# B&R Automation Studio project 8238 (part 2)

### IoMap.iom - APC2200/IoMap.iom
```iecst
(********************************************************************
 * COPYRIGHT --
 ********************************************************************
 * File: IoMap.iom
 * Author: Dave
 * Created: November 19, 2010
 ********************************************************************
 * IO mapping file
 ********************************************************************)
VAR_CONFIG
	Safety.ModuleOk AT %IX."X20SL8100".ModuleOk;
	Safety.ModuleID AT %ID."X20SL8100".ModuleID;
	Safety.FW_Version AT %ID."X20SL8100".FirmwareVersion;
	Safety.SFW_Version AT %IW."X20SL8100".SafeFirmwareVersion;
	Safety.UDID_low AT %ID."X20SL8100".UDID_low;
	Safety.UDID_high AT %IW."X20SL8100".UDID_high;
	Safety.EDM_Comm AT %QD."X20SL8100".DINT101;
	Safety.Reset_Comm AT %QD."X20SL8100".DINT102;
	Safety.MasterReset_Comm AT %QW."X20SL8100".INT1001;
	Safety.ModuleFault AT %IX."X20SL8100".BOOL00001;
	SafetyZone[1].DataFromSafePLC AT %IW."X20SL8100".INT0001;
	SafetyZone[2].DataFromSafePLC AT %IW."X20SL8100".INT0002;
	SafetyZone[3].DataFromSafePLC AT %IW."X20SL8100".INT0003;
	SafetyZone[4].DataFromSafePLC AT %IW."X20SL8100".INT0004;
	SafetyZone[5].DataFromSafePLC AT %IW."X20SL8100".INT0005;
	SafetyZone[6].DataFromSafePLC AT %IW."X20SL8100".INT0006;
	SafetyZone[7].DataFromSafePLC AT %IW."X20SL8100".INT0007;
	SafetyZone[8].DataFromSafePLC AT %IW."X20SL8100".INT0008;
	SafetyZone[9].DataFromSafePLC AT %IW."X20SL8100".INT0009;
	SafetyZone[10].DataFromSafePLC AT %IW."X20SL8100".INT0010;
	SafetyZone[11].DataFromSafePLC AT %IW."X20SL8100".INT0011;
	SafetyZone[12].DataFromSafePLC AT %IW."X20SL8100".INT0012;
	SafetyZone[13].DataFromSafePLC AT %IW."X20SL8100".INT0013;
	SafetyZone[14].DataFromSafePLC AT %IW."X20SL8100".INT0014;
	SafetyZone[15].DataFromSafePLC AT %IW."X20SL8100".INT0015;
	SafetyZone[16].DataFromSafePLC AT %IW."X20SL8100".INT0016;
	SafetyZone[17].DataFromSafePLC AT %IW."X20SL8100".INT0017;
	SafetyZone[18].DataFromSafePLC AT %IW."X20SL8100".INT0018;
	SafetyZone[19].DataFromSafePLC AT %IW."X20SL8100".INT0019;
	SafetyZone[20].DataFromSafePLC AT %IW."X20SL8100".INT0020;
	SafetyZone[21].DataFromSafePLC AT %IW."X20SL8100".INT0021;
	SafetyZone[22].DataFromSafePLC AT %IW."X20SL8100".INT0022;
	SafetyZone[23].DataFromSafePLC AT %IW."X20SL8100".INT0023;
	SafetyZone[24].DataFromSafePLC AT %IW."X20SL8100".INT0024;
	SafetyZone[25].DataFromSafePLC AT %IW."X20SL8100".INT0025;
	SafetyZone[26].DataFromSafePLC AT %IW."X20SL8100".INT0026;
	SafetyZone[27].DataFromSafePLC AT %IW."X20SL8100".INT0027;
	SafetyZone[28].DataFromSafePLC AT %IW."X20SL8100".INT0028;
	SafetyZone[29].DataFromSafePLC AT %IW."X20SL8100".INT0029;
	SafetyZone[30].DataFromSafePLC AT %IW."X20SL8100".INT0030;
	Safety.EDM_Comm AT %QD."X20SL8100".DINT1001;
	Safety.Reset_Comm AT %QD."X20SL8100".DINT1002;
	Cyclic#2.OK[1001] AT %IX."X20DM9324_1001".ModuleOk;
	Cyclic#2.OK[1002] AT %IX."X20DM9324_1002".ModuleOk;
	BusCouplerDiag[21].ModuleLostWhilstOperational AT %ID."X20BB80_400_MC01".IF1.ModuleLostWhileOperational;
	BusCouplerDiag[21].StationAtBusEnd AT %IB."X20BB80_400_MC01".IF1.StationAtBusEnd;
	BusCouplerDiag[21].StationPastOutFrameError AT %IB."X20BB80_400_MC01".IF1.StationPastOutFrameError;
	BusCouplerDiag[21].StationPastInFrameError AT %IB."X20BB80_400_MC01".IF1.StationPastInFrameError;
	BusCouplerDiag[31].ModuleLostWhilstOperational AT %ID."X67BC8321_PL31".IF1.ModuleLostWhileOperational;
	BusCouplerDiag[31].StationAtBusEnd AT %IB."X67BC8321_PL31".IF1.StationAtBusEnd;
	BusCouplerDiag[31].StationPastOutFrameError AT %IB."X67BC8321_PL31".IF1.StationPastOutFrameError;
	BusCouplerDiag[31].StationPastInFrameError AT %IB."X67BC8321_PL31".IF1.StationPastInFrameError;
	BusCouplerDiag[32].ModuleLostWhilstOperational AT %ID."X67BC8321_PL32".IF1.ModuleLostWhileOperational;
	BusCouplerDiag[32].StationAtBusEnd AT %IB."X67BC8321_PL32".IF1.StationAtBusEnd;
	BusCouplerDiag[32].StationPastOutFrameError AT %IB."X67BC8321_PL32".IF1.StationPastOutFrameError;
	BusCouplerDiag[32].StationPastInFrameError AT %IB."X67BC8321_PL32".IF1.StationPastInFrameError;
	BusCouplerDiag[33].ModuleLostWhilstOperational AT %ID."X67BC8321_PL33".IF1.ModuleLostWhileOperational;
	BusCouplerDiag[33].StationAtBusEnd AT %IB."X67BC8321_PL33".IF1.StationAtBusEnd;
	BusCouplerDiag[33].StationPastOutFrameError AT %IB."X67BC8321_PL33".IF1.StationPastOutFrameError;
	BusCouplerDiag[33].StationPastInFrameError AT %IB."X67BC8321_PL33".IF1.StationPastInFrameError;
	BusCouplerDiag[110].ModuleLostWhilstOperational AT %ID."X20BB80_400_SC01".IF1.ModuleLostWhileOperational;
	BusCouplerDiag[110].StationAtBusEnd AT %IB."X20BB80_400_SC01".IF1.StationAtBusEnd;
	BusCouplerDiag[110].StationPastOutFrameError AT %IB."X20BB80_400_SC01".IF1.StationPastOutFrameError;
	BusCouplerDiag[110].StationPastInFrameError AT %IB."X20BB80_400_SC01".IF1.StationPastInFrameError;
	Cyclic#2.ABB_EPL.Drives[11].Comm.ModuleOk AT %IX."FEPL-02_and_ACS380_SB1".ModuleOk;
	Cyclic#2.ABB_EPL.Drives[11].Comm.ErrorCode AT %IW."FEPL-02_and_ACS380_SB1".VendorSpecificAlarmCodes_I2203;
	Cyclic#2.ABB_EPL.Drives[11].Comm.ControlWord AT %QW."FEPL-02_and_ACS380_SB1".ControlWord_I6040Out;
	Cyclic#2.ABB_EPL.Drives[11].Comm.StatusWord AT %IW."FEPL-02_and_ACS380_SB1".StatusWord_I6041;
	Cyclic#2.ABB_EPL.Drives[11].Comm.TargetVelocity AT %QW."FEPL-02_and_ACS380_SB1".VlTargetVelocity_I6042Out;
	Cyclic#2.ABB_EPL.Drives[11].Comm.ActVelocity AT %IW."FEPL-02_and_ACS380_SB1".VlVelocityActualValue_I6044;
	Cyclic#2.ABB_EPL.Drives[11].Comm.ActCurrent AT %ID."FEPL-02_and_ACS380_SB1"._0107_Motor_current_I4001_S07;
	Cyclic#2.ABB_EPL.Drives[11].Comm.ActTorque AT %ID."FEPL-02_and_ACS380_SB1"._0110_Motor_torque_I4001_S0A;
	Cyclic#2.ABB_EPL.Drives[1].Comm.ModuleOk AT %IX."FEPL-02_and_ACS380_STB1".ModuleOk;
	Cyclic#2.ABB_EPL.Drives[1].Comm.ErrorCode AT %IW."FEPL-02_and_ACS380_STB1".VendorSpecificAlarmCodes_I2203;
	Cyclic#2.ABB_EPL.Drives[1].Comm.ControlWord AT %QW."FEPL-02_and_ACS380_STB1".ControlWord_I6040Out;
	Cyclic#2.ABB_EPL.Drives[1].Comm.StatusWord AT %IW."FEPL-02_and_ACS380_STB1".StatusWord_I6041;
	Cyclic#2.ABB_EPL.Drives[1].Comm.TargetVelocity AT %QW."FEPL-02_and_ACS380_STB1".VlTargetVelocity_I6042Out;
	Cyclic#2.ABB_EPL.Drives[1].Comm.ActVelocity AT %IW."FEPL-02_and_ACS380_STB1".VlVelocityActualValue_I6044;
	Cyclic#2.ABB_EPL.Drives[1].Comm.ActCurrent AT %ID."FEPL-02_and_ACS380_STB1"._0107_Motor_current_I4001_S07;
	Cyclic#2.ABB_EPL.Drives[1].Comm.ActTorque AT %ID."FEPL-02_and_ACS380_STB1"._0110_Motor_torque_I4001_S0A;
	Cyclic#2.ABB_EPL.Drives[12].Comm.ModuleOk AT %IX."FEPL-02_and_ACS380_SB2".ModuleOk;
	Cyclic#2.ABB_EPL.Drives[12].Comm.ErrorCode AT %IW."FEPL-02_and_ACS380_SB2".VendorSpecificAlarmCodes_I2203;
	Cyclic#2.ABB_EPL.Drives[12].Comm.ControlWord AT %QW."FEPL-02_and_ACS380_SB2".ControlWord_I6040Out;
	Cyclic#2.ABB_EPL.Drives[12].Comm.StatusWord AT %IW."FEPL-02_and_ACS380_SB2".StatusWord_I6041;
	Cyclic#2.ABB_EPL.Drives[12].Comm.TargetVelocity AT %QW."FEPL-02_and_ACS380_SB2".VlTargetVelocity_I6042Out;
	Cyclic#2.ABB_EPL.Drives[12].Comm.ActVelocity AT %IW."FEPL-02_and_ACS380_SB2".VlVelocityActualValue_I6044;
	Cyclic#2.ABB_EPL.Drives[12].Comm.ActCurrent AT %ID."FEPL-02_and_ACS380_SB2"._0107_Motor_current_I4001_S07;
	Cyclic#2.ABB_EPL.Drives[12].Comm.ActTorque AT %ID."FEPL-02_and_ACS380_SB2"._0110_Motor_torque_I4001_S0A;
	Cyclic#2.ABB_EPL.Drives[2].Comm.ModuleOk AT %IX."FEPL-02_and_ACS380_STB2".ModuleOk;
	Cyclic#2.ABB_EPL.Drives[2].Comm.ErrorCode AT %IW."FEPL-02_and_ACS380_STB2".VendorSpecificAlarmCodes_I2203;
	Cyclic#2.ABB_EPL.Drives[2].Comm.ControlWord AT %QW."FEPL-02_and_ACS380_STB2".ControlWord_I6040Out;
	Cyclic#2.ABB_EPL.Drives[2].Comm.StatusWord AT %IW."FEPL-02_and_ACS380_STB2".StatusWord_I6041;
	Cyclic#2.ABB_EPL.Drives[2].Comm.TargetVelocity AT %QW."FEPL-02_and_ACS380_STB2".VlTargetVelocity_I6042Out;
	Cyclic#2.ABB_EPL.Drives[2].Comm.ActVelocity AT %IW."FEPL-02_and_ACS380_STB2".VlVelocityActualValue_I6044;
	Cyclic#2.ABB_EPL.Drives[2].Comm.ActCurrent AT %ID."FEPL-02_and_ACS380_STB2"._0107_Motor_current_I4001_S07;
	Cyclic#2.ABB_EPL.Drives[2].Comm.ActTorque AT %ID."FEPL-02_and_ACS380_STB2"._0110_Motor_torque_I4001_S0A;
	SM[1401].ModuleOk AT %IX."X67SI8103_1401".ModuleOk;
	SM[1401].ModuleID AT %IW."X67SI8103_1401".ModuleID;
	SM[1401].HardwareVariant AT %IW."X67SI8103_1401".HardwareVariant;
	SM[1401].FirmwareVersion AT %IW."X67SI8103_1401".FirmwareVersion;
	SM[1401].SafeModuleOK AT %IX."X67SI8103_1401".SafeModuleOK;
	SM[1401].SafeDigitialInput01 AT %IX."X67SI8103_1401".SafeDigitalInput01;
	SM[1401].SafeDigitialInput02 AT %IX."X67SI8103_1401".SafeDigitalInput02;
	SM[1401].SafeDigitialInput03 AT %IX."X67SI8103_1401".SafeDigitalInput03;
	SM[1401].SafeDigitialInput04 AT %IX."X67SI8103_1401".SafeDigitalInput04;
	SM[1401].SafeDigitialInput05 AT %IX."X67SI8103_1401".SafeDigitalInput05;
	SM[1401].SafeDigitialInput06 AT %IX."X67SI8103_1401".SafeDigitalInput06;
	SM[1401].SafeDigitialInput07 AT %IX."X67SI8103_1401".SafeDigitalInput07;
	SM[1401].SafeDigitialInput08 AT %IX."X67SI8103_1401".SafeDigitalInput08;
	SM[1401].SafeTwoChannelInput0102 AT %IX."X67SI8103_1401".SafeTwoChannelInput0102;
	SM[1401].SafeTwoChannelInput0304 AT %IX."X67SI8103_1401".SafeTwoChannelInput0304;
	SM[1401].SafeTwoChannelInput0506 AT %IX."X67SI8103_1401".SafeTwoChannelInput0506;
	SM[1401].SafeTwoChannelInput0708 AT %IX."X67SI8103_1401".SafeTwoChannelInput0708;
	SM[1401].SafeTwoChannelOk0102 AT %IX."X67SI8103_1401".SafeTwoChannelOK0102;
	SM[1401].SafeTwoChannelOk0304 AT %IX."X67SI8103_1401".SafeTwoChannelOK0304;
	SM[1401].SafeTwoChannelOk0506 AT %IX."X67SI8103_1401".SafeTwoChannelOK0506;
	SM[1401].SafeTwoChannelOk0708 AT %IX."X67SI8103_1401".SafeTwoChannelOK0708;
	SM[1401].DigitalInput01 AT %IX."X67SI8103_1401".DigitalInput01;
	SM[1401].DigitalInput02 AT %IX."X67SI8103_1401".DigitalInput02;
	SM[1401].DigitalOutput01 AT %QX."X67SI8103_1401".DigitalOutput01;
	SM[1401].DigitalOutput02 AT %QX."X67SI8103_1401".DigitalOutput02;
	SM[1402].ModuleOk AT %IX."X67SI8103_1402".ModuleOk;
	SM[1402].ModuleID AT %IW."X67SI8103_1402".ModuleID;
	SM[1402].HardwareVariant AT %IW."X67SI8103_1402".HardwareVariant;
	SM[1402].FirmwareVersion AT %IW."X67SI8103_1402".FirmwareVersion;
	SM[1402].SafeModuleOK AT %IX."X67SI8103_1402".SafeModuleOK;
	SM[1402].SafeDigitialInput01 AT %IX."X67SI8103_1402".SafeDigitalInput01;
	SM[1402].SafeDigitialInput02 AT %IX."X67SI8103_1402".SafeDigitalInput02;
	SM[1402].SafeDigitialInput03 AT %IX."X67SI8103_1402".SafeDigitalInput03;
	SM[1402].SafeDigitialInput04 AT %IX."X67SI8103_1402".SafeDigitalInput04;
	SM[1402].SafeDigitialInput05 AT %IX."X67SI8103_1402".SafeDigitalInput05;
	SM[1402].SafeDigitialInput06 AT %IX."X67SI8103_1402".SafeDigitalInput06;
	SM[1402].SafeDigitialInput07 AT %IX."X67SI8103_1402".SafeDigitalInput07;
	SM[1402].SafeDigitialInput08 AT %IX."X67SI8103_1402".SafeDigitalInput08;
	SM[1402].SafeTwoChannelInput0102 AT %IX."X67SI8103_1402".SafeTwoChannelInput0102;
	SM[1402].SafeTwoChannelInput0304 AT %IX."X67SI8103_1402".SafeTwoChannelInput0304;
	SM[1402].SafeTwoChannelInput0506 AT %IX."X67SI8103_1402".SafeTwoChannelInput0506;
	SM[1402].SafeTwoChannelInput0708 AT %IX."X67SI8103_1402".SafeTwoChannelInput0708;
	SM[1402].SafeTwoChannelOk0102 AT %IX."X67SI8103_1402".SafeTwoChannelOK0102;
	SM[1402].SafeTwoChannelOk0304 AT %IX."X67SI8103_1402".SafeTwoChannelOK0304;
	SM[1402].SafeTwoChannelOk0506 AT %IX."X67SI8103_1402".SafeTwoChannelOK0506;
	SM[1402].SafeTwoChannelOk0708 AT %IX."X67SI8103_1402".SafeTwoChannelOK0708;
	SM[1402].DigitalInput01 AT %IX."X67SI8103_1402".DigitalInput01;
	SM[1402].DigitalInput02 AT %IX."X67SI8103_1402".DigitalInput02;
	SM[1402].DigitalOutput01 AT %QX."X67SI8103_1402".DigitalOutput01;
	SM[1402].DigitalOutput02 AT %QX."X67SI8103_1402".DigitalOutput02;
	SM[1403].ModuleOk AT %IX."X67SI8103_1403".ModuleOk;
	SM[1403].ModuleID AT %IW."X67SI8103_1403".ModuleID;
	SM[1403].HardwareVariant AT %IW."X67SI8103_1403".HardwareVariant;
	SM[1403].FirmwareVersion AT %IW."X67SI8103_1403".FirmwareVersion;
	SM[1403].SafeModuleOK AT %IX."X67SI8103_1403".SafeModuleOK;
	SM[1403].SafeDigitialInput01 AT %IX."X67SI8103_1403".SafeDigitalInput01;
	SM[1403].SafeDigitialInput02 AT %IX."X67SI8103_1403".SafeDigitalInput02;
	SM[1403].SafeDigitialInput03 AT %IX."X67SI8103_1403".SafeDigitalInput03;
	SM[1403].SafeDigitialInput04 AT %IX."X67SI8103_1403".SafeDigitalInput04;
	SM[1403].SafeDigitialInput05 AT %IX."X67SI8103_1403".SafeDigitalInput05;
	SM[1403].SafeDigitialInput06 AT %IX."X67SI8103_1403".SafeDigitalInput06;
	SM[1403].SafeDigitialInput07 AT %IX."X67SI8103_1403".SafeDigitalInput07;
	SM[1403].SafeDigitialInput08 AT %IX."X67SI8103_1403".SafeDigitalInput08;
	SM[1403].SafeTwoChannelInput0102 AT %IX."X67SI8103_1403".SafeTwoChannelInput0102;
	SM[1403].SafeTwoChannelInput0304 AT %IX."X67SI8103_1403".SafeTwoChannelInput0304;
	SM[1403].SafeTwoChannelInput0506 AT %IX."X67SI8103_1403".SafeTwoChannelInput0506;
	SM[1403].SafeTwoChannelInput0708 AT %IX."X67SI8103_1403".SafeTwoChannelInput0708;
	SM[1403].SafeTwoChannelOk0102 AT %IX."X67SI8103_1403".SafeTwoChannelOK0102;
	SM[1403].SafeTwoChannelOk0304 AT %IX."X67SI8103_1403".SafeTwoChannelOK0304;
	SM[1403].SafeTwoChannelOk0506 AT %IX."X67SI8103_1403".SafeTwoChannelOK0506;
	SM[1403].SafeTwoChannelOk0708 AT %IX."X67SI8103_1403".SafeTwoChannelOK0708;
	SM[1403].DigitalInput01 AT %IX."X67SI8103_1403".DigitalInput01;
	SM[1403].DigitalInput02 AT %IX."X67SI8103_1403".DigitalInput02;
	SM[1403].DigitalOutput01 AT %QX."X67SI8103_1403".DigitalOutput01;
	SM[1403].DigitalOutput02 AT %QX."X67SI8103_1403".DigitalOutput02;
	SM[1406].ModuleOk AT %IX."X67SI8103_1406".ModuleOk;
	SM[1406].ModuleID AT %IW."X67SI8103_1406".ModuleID;
	SM[1406].HardwareVariant AT %IW."X67SI8103_1406".HardwareVariant;
	SM[1406].FirmwareVersion AT %IW."X67SI8103_1406".FirmwareVersion;
	SM[1406].SafeModuleOK AT %IX."X67SI8103_1406".SafeModuleOK;
	SM[1406].SafeDigitialInput01 AT %IX."X67SI8103_1406".SafeDigitalInput01;
	SM[1406].SafeDigitialInput02 AT %IX."X67SI8103_1406".SafeDigitalInput02;
	SM[1406].SafeDigitialInput03 AT %IX."X67SI8103_1406".SafeDigitalInput03;
	SM[1406].SafeDigitialInput04 AT %IX."X67SI8103_1406".SafeDigitalInput04;
	SM[1406].SafeDigitialInput05 AT %IX."X67SI8103_1406".SafeDigitalInput05;
	SM[1406].SafeDigitialInput06 AT %IX."X67SI8103_1406".SafeDigitalInput06;
	SM[1406].SafeDigitialInput07 AT %IX."X67SI8103_1406".SafeDigitalInput07;
	SM[1406].SafeDigitialInput08 AT %IX."X67SI8103_1406".SafeDigitalInput08;
	SM[1406].SafeTwoChannelInput0102 AT %IX."X67SI8103_1406".SafeTwoChannelInput0102;
	SM[1406].SafeTwoChannelInput0304 AT %IX."X67SI8103_1406".SafeTwoChannelInput0304;
	SM[1406].SafeTwoChannelInput0506 AT %IX."X67SI8103_1406".SafeTwoChannelInput0506;
	SM[1406].SafeTwoChannelInput0708 AT %IX."X67SI8103_1406".SafeTwoChannelInput0708;
	SM[1406].SafeTwoChannelOk0102 AT %IX."X67SI8103_1406".SafeTwoChannelOK0102;
	SM[1406].SafeTwoChannelOk0304 AT %IX."X67SI8103_1406".SafeTwoChannelOK0304;
	SM[1406].SafeTwoChannelOk0506 AT %IX."X67SI8103_1406".SafeTwoChannelOK0506;
	SM[1406].SafeTwoChannelOk0708 AT %IX."X67SI8103_1406".SafeTwoChannelOK0708;
	SM[1406].DigitalInput01 AT %IX."X67SI8103_1406".DigitalInput01;
	SM[1406].DigitalInput02 AT %IX."X67SI8103_1406".DigitalInput02;
	SM[1406].DigitalOutput01 AT %QX."X67SI8103_1406".DigitalOutput01;
	SM[1406].DigitalOutput02 AT %QX."X67SI8103_1406".DigitalOutput02;
	WeightRaw[1349].Wgt_Channel_1 AT %ID."X67AI2744_1801".AnalogInput01;
	WeightRaw[1352].Wgt_Channel_1 AT %ID."X67AI2744_1802".AnalogInput01;
	WeightRaw[1355].Wgt_Channel_1 AT %ID."X67AI2744_1803".AnalogInput01;
	SM[1410].ModuleOk AT %IX."X67SI8103_1410".ModuleOk;
	SM[1410].ModuleID AT %IW."X67SI8103_1410".ModuleID;
	SM[1410].HardwareVariant AT %IW."X67SI8103_1410".HardwareVariant;
	SM[1410].FirmwareVersion AT %IW."X67SI8103_1410".FirmwareVersion;
	SM[1410].SafeModuleOK AT %IX."X67SI8103_1410".SafeModuleOK;
	SM[1410].SafeDigitialInput01 AT %IX."X67SI8103_1410".SafeDigitalInput01;
	SM[1410].SafeDigitialInput02 AT %IX."X67SI8103_1410".SafeDigitalInput02;
	SM[1410].SafeDigitialInput03 AT %IX."X67SI8103_1410".SafeDigitalInput03;
	SM[1410].SafeDigitialInput04 AT %IX."X67SI8103_1410".SafeDigitalInput04;
	SM[1410].SafeDigitialInput05 AT %IX."X67SI8103_1410".SafeDigitalInput05;
	SM[1410].SafeDigitialInput06 AT %IX."X67SI8103_1410".SafeDigitalInput06;
	SM[1410].SafeDigitialInput07 AT %IX."X67SI8103_1410".SafeDigitalInput07;
	SM[1410].SafeDigitialInput08 AT %IX."X67SI8103_1410".SafeDigitalInput08;
	SM[1410].SafeTwoChannelInput0102 AT %IX."X67SI8103_1410".SafeTwoChannelInput0102;
	SM[1410].SafeTwoChannelInput0304 AT %IX."X67SI8103_1410".SafeTwoChannelInput0304;
	SM[1410].SafeTwoChannelInput0506 AT %IX."X67SI8103_1410".SafeTwoChannelInput0506;
	SM[1410].SafeTwoChannelInput0708 AT %IX."X67SI8103_1410".SafeTwoChannelInput0708;
	SM[1410].SafeTwoChannelOk0102 AT %IX."X67SI8103_1410".SafeTwoChannelOK0102;
	SM[1410].SafeTwoChannelOk0304 AT %IX."X67SI8103_1410".SafeTwoChannelOK0304;
	SM[1410].SafeTwoChannelOk0506 AT %IX."X67SI8103_1410".SafeTwoChannelOK0506;
	SM[1410].SafeTwoChannelOk0708 AT %IX."X67SI8103_1410".SafeTwoChannelOK0708;
	SM[1410].DigitalInput01 AT %IX."X67SI8103_1410".DigitalInput01;
	SM[1410].DigitalInput02 AT %IX."X67SI8103_1410".DigitalInput02;
	SM[1410].DigitalOutput01 AT %QX."X67SI8103_1410".DigitalOutput01;
	SM[1410].DigitalOutput02 AT %QX."X67SI8103_1410".DigitalOutput02;
	SM[1411].ModuleOk AT %IX."X67SI8103_1411".ModuleOk;
	SM[1411].ModuleID AT %IW."X67SI8103_1411".ModuleID;
	SM[1411].HardwareVariant AT %IW."X67SI8103_1411".HardwareVariant;
	SM[1411].FirmwareVersion AT %IW."X67SI8103_1411".FirmwareVersion;
	SM[1411].SafeModuleOK AT %IX."X67SI8103_1411".SafeModuleOK;
	SM[1411].SafeDigitialInput01 AT %IX."X67SI8103_1411".SafeDigitalInput01;
	SM[1411].SafeDigitialInput02 AT %IX."X67SI8103_1411".SafeDigitalInput02;
	SM[1411].SafeDigitialInput03 AT %IX."X67SI8103_1411".SafeDigitalInput03;
	SM[1411].SafeDigitialInput04 AT %IX."X67SI8103_1411".SafeDigitalInput04;
	SM[1411].SafeDigitialInput05 AT %IX."X67SI8103_1411".SafeDigitalInput05;
	SM[1411].SafeDigitialInput06 AT %IX."X67SI8103_1411".SafeDigitalInput06;
	SM[1411].SafeDigitialInput07 AT %IX."X67SI8103_1411".SafeDigitalInput07;
	SM[1411].SafeDigitialInput08 AT %IX."X67SI8103_1411".SafeDigitalInput08;
	SM[1411].SafeTwoChannelInput0102 AT %IX."X67SI8103_1411".SafeTwoChannelInput0102;
	SM[1411].SafeTwoChannelInput0304 AT %IX."X67SI8103_1411".SafeTwoChannelInput0304;
	SM[1411].SafeTwoChannelInput0506 AT %IX."X67SI8103_1411".SafeTwoChannelInput0506;
	SM[1411].SafeTwoChannelInput0708 AT %IX."X67SI8103_1411".SafeTwoChannelInput0708;
	SM[1411].SafeTwoChannelOk0102 AT %IX."X67SI8103_1411".SafeTwoChannelOK0102;
	SM[1411].SafeTwoChannelOk0304 AT %IX."X67SI8103_1411".SafeTwoChannelOK0304;
	SM[1411].SafeTwoChannelOk0506 AT %IX."X67SI8103_1411".SafeTwoChannelOK0506;
	SM[1411].SafeTwoChannelOk0708 AT %IX."X67SI8103_1411".SafeTwoChannelOK0708;
	SM[1411].DigitalInput01 AT %IX."X67SI8103_1411".DigitalInput01;
	SM[1411].DigitalInput02 AT %IX."X67SI8103_1411".DigitalInput02;
	SM[1411].DigitalOutput01 AT %QX."X67SI8103_1411".DigitalOutput01;
	SM[1411].DigitalOutput02 AT %QX."X67SI8103_1411".DigitalOutput02;
	SM[1416].ModuleOk AT %IX."X67SI8103_1416".ModuleOk;
	SM[1416].ModuleID AT %IW."X67SI8103_1416".ModuleID;
	SM[1416].HardwareVariant AT %IW."X67SI8103_1416".HardwareVariant;
	SM[1416].FirmwareVersion AT %IW."X67SI8103_1416".FirmwareVersion;
	SM[1416].SafeModuleOK AT %IX."X67SI8103_1416".SafeModuleOK;
	SM[1416].SafeDigitialInput01 AT %IX."X67SI8103_1416".SafeDigitalInput01;
	SM[1416].SafeDigitialInput02 AT %IX."X67SI8103_1416".SafeDigitalInput02;
	SM[1416].SafeDigitialInput03 AT %IX."X67SI8103_1416".SafeDigitalInput03;
	SM[1416].SafeDigitialInput04 AT %IX."X67SI8103_1416".SafeDigitalInput04;
	SM[1416].SafeDigitialInput05 AT %IX."X67SI8103_1416".SafeDigitalInput05;
	SM[1416].SafeDigitialInput06 AT %IX."X67SI8103_1416".SafeDigitalInput06;
	SM[1416].SafeDigitialInput07 AT %IX."X67SI8103_1416".SafeDigitalInput07;
	SM[1416].SafeDigitialInput08 AT %IX."X67SI8103_1416".SafeDigitalInput08;
	SM[1416].SafeTwoChannelInput0102 AT %IX."X67SI8103_1416".SafeTwoChannelInput0102;
	SM[1416].SafeTwoChannelInput0304 AT %IX."X67SI8103_1416".SafeTwoChannelInput0304;
	SM[1416].SafeTwoChannelInput0506 AT %IX."X67SI8103_1416".SafeTwoChannelInput0506;
	SM[1416].SafeTwoChannelInput0708 AT %IX."X67SI8103_1416".SafeTwoChannelInput0708;
	SM[1416].SafeTwoChannelOk0102 AT %IX."X67SI8103_1416".SafeTwoChannelOK0102;
	SM[1416].SafeTwoChannelOk0304 AT %IX."X67SI8103_1416".SafeTwoChannelOK0304;
	SM[1416].SafeTwoChannelOk0506 AT %IX."X67SI8103_1416".SafeTwoChannelOK0506;
	SM[1416].SafeTwoChannelOk0708 AT %IX."X67SI8103_1416".SafeTwoChannelOK0708;
	SM[1416].DigitalInput01 AT %IX."X67SI8103_1416".DigitalInput01;
	SM[1416].DigitalInput02 AT %IX."X67SI8103_1416".DigitalInput02;
	SM[1416].DigitalOutput01 AT %QX."X67SI8103_1416".DigitalOutput01;
	SM[1416].DigitalOutput02 AT %QX."X67SI8103_1416".DigitalOutput02;
	BusCouplerDiag[34].ModuleLostWhilstOperational AT %ID."X67BC8321_PL34".IF1.ModuleLostWhileOperational;
	BusCouplerDiag[34].StationAtBusEnd AT %IB."X67BC8321_PL34".IF1.StationAtBusEnd;
	BusCouplerDiag[34].StationPastOutFrameError AT %IB."X67BC8321_PL34".IF1.StationPastOutFrameError;
	BusCouplerDiag[34].StationPastInFrameError AT %IB."X67BC8321_PL34".IF1.StationPastInFrameError;
	BusCouplerDiag[35].ModuleLostWhilstOperational AT %ID."X67BC8321_PL35".IF1.ModuleLostWhileOperational;
	BusCouplerDiag[35].StationAtBusEnd AT %IB."X67BC8321_PL35".IF1.StationAtBusEnd;
	BusCouplerDiag[35].StationPastOutFrameError AT %IB."X67BC8321_PL35".IF1.StationPastOutFrameError;
	BusCouplerDiag[35].StationPastInFrameError AT %IB."X67BC8321_PL35".IF1.StationPastInFrameError;
	BusCouplerDiag[41].ModuleLostWhilstOperational AT %ID."X67BC8321_PL36".IF1.ModuleLostWhileOperational;
	BusCouplerDiag[42].ModuleLostWhilstOperational AT %ID."X67BC8321_PL37".IF1.ModuleLostWhileOperational;
	BusCouplerDiag[43].ModuleLostWhilstOperational AT %ID."X67BC8321_PL38".IF1.ModuleLostWhileOperational;
	BusCouplerDiag[44].ModuleLostWhilstOperational AT %ID."X67BC8321_PL39".IF1.ModuleLostWhileOperational;
	BusCouplerDiag[41].StationAtBusEnd AT %IB."X67BC8321_PL36".IF1.StationAtBusEnd;
	BusCouplerDiag[42].StationAtBusEnd AT %IB."X67BC8321_PL37".IF1.StationAtBusEnd;
	BusCouplerDiag[41].StationPastOutFrameError AT %IB."X67BC8321_PL36".IF1.StationPastOutFrameError;
	BusCouplerDiag[42].StationPastOutFrameError AT %IB."X67BC8321_PL37".IF1.StationPastOutFrameError;
	BusCouplerDiag[42].StationPastInFrameError AT %IB."X67BC8321_PL37".IF1.StationPastInFrameError;
	BusCouplerDiag[41].StationPastInFrameError AT %IB."X67BC8321_PL36".IF1.StationPastInFrameError;
	BusCouplerDiag[44].StationPastInFrameError AT %IB."X67BC8321_PL39".IF1.StationPastInFrameError;
	BusCouplerDiag[44].StationPastOutFrameError AT %IB."X67BC8321_PL39".IF1.StationPastOutFrameError;
	BusCouplerDiag[44].StationAtBusEnd AT %IB."X67BC8321_PL39".IF1.StationAtBusEnd;
	BusCouplerDiag[43].StationAtBusEnd AT %IB."X67BC8321_PL38".IF1.StationAtBusEnd;
	BusCouplerDiag[43].StationPastOutFrameError AT %IB."X67BC8321_PL38".IF1.StationPastOutFrameError;
	BusCouplerDiag[43].StationPastInFrameError AT %IB."X67BC8321_PL38".IF1.StationPastInFrameError;
	Cyclic#2.X[1001].X01 AT %IX."X20DM9324_1001".DigitalInput01; (*spare*) (*spare*)
	Cyclic#2.Y[1001].Y01 AT %QX."X20DM9324_1001".DigitalOutput01; (*Light Tower Green*) (*SafetyZone[1].TowerLight.TL_DO_Green*)
	Cyclic#2.X[1001].X02 AT %IX."X20DM9324_1001".DigitalInput02; (*Air pressure switch*) (*SafetyZone[1].PressureSwitch*)
	Cyclic#2.Y[1001].Y02 AT %QX."X20DM9324_1001".DigitalOutput02; (*Light Tower Yellow*) (*SafetyZone[1].TowerLight.TL_DO_Yellow*)
	Cyclic#2.X[1001].X03 AT %IX."X20DM9324_1001".DigitalInput03; (*Safety Reset button*) (*MasterReset_1*)
	Cyclic#2.Y[1001].Y03 AT %QX."X20DM9324_1001".DigitalOutput03; (*Light Tower Red*) (*SafetyZone[1].TowerLight.TL_DO_Red*)
	Cyclic#2.X[1001].X04 AT %IX."X20DM9324_1001".DigitalInput04; (*Fuse Reset*) (*Fuse_Reset_1*)
	Cyclic#2.Y[1001].Y04 AT %QX."X20DM9324_1001".DigitalOutput04; (*Light Tower Siren*) (*SafetyZone[1].TowerLight.TL_DO_Sounder*)
	Cyclic#2.X[1001].X05 AT %IX."X20DM9324_1001".DigitalInput05; (*spare*) (*spare*)
	Cyclic#2.X[1001].X06 AT %IX."X20DM9324_1001".DigitalInput06; (*spare*) (*spare*)
	Cyclic#2.X[1001].X07 AT %IX."X20DM9324_1001".DigitalInput07; (*spare*) (*spare*)
	Cyclic#2.X[1001].X08 AT %IX."X20DM9324_1001".DigitalInput08; (*spare*) (*spare*)
	Cyclic#2.X[1002].X01 AT %IX."X20DM9324_1002".DigitalInput01; (*Safety Relay D1.1 Monitor*) (*SafetyZone[2].EDM*)
	Cyclic#2.Y[1002].Y01 AT %QX."X20DM9324_1002".DigitalOutput01; (*Safety Reset Button Lamp*) (*SafetyZone[1].Main_Lamp*)
	Cyclic#2.X[1002].X02 AT %IX."X20DM9324_1002".DigitalInput02; (*Safety Relay D2.1 Monitor*) (*SafetyZone[3].EDM*)
	Cyclic#2.Y[1002].Y02 AT %QX."X20DM9324_1002".DigitalOutput02; (*Fuse Reset Button*) (*Fuse_Lamp_1*)
	Cyclic#2.X[1002].X03 AT %IX."X20DM9324_1002".DigitalInput03; (*Safety Relay D3.1 Monitor*) (*SafetyZone[4].EDM*)
	Cyclic#2.Y[1002].Y03 AT %QX."X20DM9324_1002".DigitalOutput03; (*spare*) (*spare*)
	Cyclic#2.X[1002].X04 AT %IX."X20DM9324_1002".DigitalInput04; (*Safety Relay D4.1 Monitor*) (*SafetyZone[5].EDM*)
	Cyclic#2.Y[1002].Y04 AT %QX."X20DM9324_1002".DigitalOutput04; (*spare*) (*spare*)
	Cyclic#2.X[1002].X05 AT %IX."X20DM9324_1002".DigitalInput05; (*spare*) (*spare*)
	Cyclic#2.X[1002].X06 AT %IX."X20DM9324_1002".DigitalInput06; (*spare*) (*spare*)
	Cyclic#2.X[1002].X07 AT %IX."X20DM9324_1002".DigitalInput07; (*spare*) (*spare*)
	Cyclic#2.X[1002].X08 AT %IX."X20DM9324_1002".DigitalInput08; (*spare*) (*spare*)
	Cyclic#2.OK[1302] AT %IX."X67DM1321_1302".ModuleOk;
	Cyclic#2.OK[1304] AT %IX."X67DM1321_1304".ModuleOk;
	Cyclic#2.OK[1306] AT %IX."X67DM1321_1306".ModuleOk;
	Cyclic#2.OK[1308] AT %IX."X67DM1321_1308".ModuleOk;
	Cyclic#2.OK[1310] AT %IX."X67DM1321_1310".ModuleOk;
	Cyclic#2.OK[1312] AT %IX."X67DM1321_1312".ModuleOk;
	Cyclic#2.OK[1314] AT %IX."X67DM1321_1314".ModuleOk;
	Cyclic#2.OK[1316] AT %IX."X67DM1321_1316".ModuleOk;
	Cyclic#2.OK[1318] AT %IX."X67DM1321_1318".ModuleOk;
	Cyclic#2.OK[1320] AT %IX."X67DM1321_1320".ModuleOk;
	Cyclic#2.OK[1319] AT %IX."X67DM1321_1319".ModuleOk;
	Cyclic#2.OK[1317] AT %IX."X67DM1321_1317".ModuleOk;
	Cyclic#2.OK[1315] AT %IX."X67DM1321_1315".ModuleOk;
	Cyclic#2.OK[1313] AT %IX."X67DM1321_1313".ModuleOk;
	Cyclic#2.OK[1311] AT %IX."X67DM1321_1311".ModuleOk;
	Cyclic#2.OK[1309] AT %IX."X67DM1321_1309".ModuleOk;
	Cyclic#2.OK[1307] AT %IX."X67DM1321_1307".ModuleOk;
	Cyclic#2.OK[1305] AT %IX."X67DM1321_1305".ModuleOk;
	Cyclic#2.OK[1303] AT %IX."X67DM1321_1303".ModuleOk;
	Cyclic#2.OK[1301] AT %IX."X67DM1321_1301".ModuleOk;
	Cyclic#2.OK[1352] AT %IX."X67DM1321_1352".ModuleOk;
	Cyclic#2.OK[1501] AT %IX."X67DM1321_1501".ModuleOk;
	Cyclic#2.OK[1502] AT %IX."X67DM1321_1502".ModuleOk;
	Cyclic#2.OK[1349] AT %IX."X67DM1321_1349".ModuleOk;
	Cyclic#2.OK[1510] AT %IX."X67DM1321_1510".ModuleOk;
	Cyclic#2.OK[1511] AT %IX."X67DM1321_1511".ModuleOk;
	Cyclic#2.OK[2514] AT %IX."X67DM1321_1508".ModuleOk;
	OK[1351] AT %IX."X67DM1321_1351".ModuleOk;
	OK[1354] AT %IX."X67DM1321_1354".ModuleOk;
	OK[1355] AT %IX."X67DM1321_1355".ModuleOk;
	OK[1357] AT %IX."X67DM1321_1357".ModuleOk;
	OK[1358] AT %IX."X67DM1321_1358".ModuleOk;
	OK[1360] AT %IX."X67DM1321_1360".ModuleOk;
	OK[1361] AT %IX."X67DM1321_1361".ModuleOk;
	OK[1363] AT %IX."X67DM1321_1363".ModuleOk;
	OK[1364] AT %IX."X67DM1321_1364".ModuleOk;
	OK[1366] AT %IX."X67DM1321_1366".ModuleOk;
	OK[1367] AT %IX."X67DM1321_1367".ModuleOk;
	WeightRaw[1358].Wgt_Channel_1 AT %ID."X67AI2744_1804".AnalogInput01;
	WeightRaw[1361].Wgt_Channel_1 AT %ID."X67AI2744_1805".AnalogInput01;
	WeightRaw[1364].Wgt_Channel_1 AT %ID."X67AI2744_1806".AnalogInput01;
	OK[1369] AT %IX."X67DM1321_1369".ModuleOk;
	WeightRaw[1367].Wgt_Channel_1 AT %ID."X67AI2744_1807".AnalogInput01;
	OK[1370] AT %IX."X67DM1321_1370".ModuleOk;
	OK[1372] AT %IX."X67DM1321_1372".ModuleOk;
	WeightRaw[1370].Wgt_Channel_1 AT %ID."X67AI2744_1808".AnalogInput01;
	OK[1373] AT %IX."X67DM1321_1373".ModuleOk;
	OK[1375] AT %IX."X67DM1321_1375".ModuleOk;
	WeightRaw[1373].Wgt_Channel_1 AT %ID."X67AI2744_1809".AnalogInput01;
	OK[1376] AT %IX."X67DM1321_1376".ModuleOk;
	OK[1378] AT %IX."X67DM1321_1378".ModuleOk;
	WeightRaw[1376].Wgt_Channel_1 AT %ID."X67AI2744_1810".AnalogInput01;
	OK[1379] AT %IX."X67DM1321_1379".ModuleOk;
	OK[1381] AT %IX."X67DM1321_1381".ModuleOk;
	WeightRaw[1379].Wgt_Channel_1 AT %ID."X67AI2744_1811".AnalogInput01;
	OK[1382] AT %IX."X67DM1321_1382".ModuleOk;
	OK[1384] AT %IX."X67DM1321_1384".ModuleOk;
	WeightRaw[1382].Wgt_Channel_1 AT %ID."X67AI2744_1812".AnalogInput01;
	OK[1385] AT %IX."X67DM1321_1385".ModuleOk;
	OK[1387] AT %IX."X67DM1321_1387".ModuleOk;
	WeightRaw[1385].Wgt_Channel_1 AT %ID."X67AI2744_1813".AnalogInput01;
	OK[1388] AT %IX."X67DM1321_1388".ModuleOk;
	OK[1390] AT %IX."X67DM1321_1390".ModuleOk;
	WeightRaw[1388].Wgt_Channel_1 AT %ID."X67AI2744_1814".AnalogInput01;
	OK[1391] AT %IX."X67DM1321_1391".ModuleOk;
	OK[1393] AT %IX."X67DM1321_1393".ModuleOk;
	WeightRaw[1391].Wgt_Channel_1 AT %ID."X67AI2744_1815".AnalogInput01;
	OK[1394] AT %IX."X67DM1321_1394".ModuleOk;
	OK[1396] AT %IX."X67DM1321_1396".ModuleOk;
	WeightRaw[1394].Wgt_Channel_1 AT %ID."X67AI2744_1816".AnalogInput01;
	OK[1397] AT %IX."X67DM1321_1397".ModuleOk;
	OK[1399] AT %IX."X67DM1321_1399".ModuleOk;
	WeightRaw[1397].Wgt_Channel_1 AT %ID."X67AI2744_1817".AnalogInput01;
	OK[1600] AT %IX."X67DM1321_1600".ModuleOk;
	OK[1602] AT %IX."X67DM1321_1602".ModuleOk;
	WeightRaw[1600].Wgt_Channel_1 AT %ID."X67AI2744_1818".AnalogInput01;
	OK[1603] AT %IX."X67DM1321_1603".ModuleOk;
	OK[1605] AT %IX."X67DM1321_1605".ModuleOk;
	WeightRaw[1603].Wgt_Channel_1 AT %ID."X67AI2744_1819".AnalogInput01;
	OK[1606] AT %IX."X67DM1321_1606".ModuleOk;
	OK[1608] AT %IX."X67DM1321_1608".ModuleOk;
	WeightRaw[1606].Wgt_Channel_1 AT %ID."X67AI2744_1820".AnalogInput01;
	OK[1609] AT %IX."X67DM1321_1609".ModuleOk;
	OK[1611] AT %IX."X67DM1321_1611".ModuleOk;
	WeightRaw[1609].Wgt_Channel_1 AT %ID."X67AI2744_1821".AnalogInput01;
	OK[1612] AT %IX."X67DM1321_1612".ModuleOk;
	OK[1614] AT %IX."X67DM1321_1614".ModuleOk;
	WeightRaw[1612].Wgt_Channel_1 AT %ID."X67AI2744_1822".AnalogInput01;
	OK[1615] AT %IX."X67DM1321_1615".ModuleOk;
	OK[1617] AT %IX."X67DM1321_1617".ModuleOk;
	WeightRaw[1615].Wgt_Channel_1 AT %ID."X67AI2744_1823".AnalogInput01;
	OK[1618] AT %IX."X67DM1321_1618".ModuleOk;
	OK[1620] AT %IX."X67DM1321_1620".ModuleOk;
	WeightRaw[1618].Wgt_Channel_1 AT %ID."X67AI2744_1824".AnalogInput01;
	WeightRaw[1301].Wgt_Channel_1 AT %ID."X67AI2744_1825".AnalogInput01;
	WeightRaw[1303].Wgt_Channel_1 AT %ID."X67AI2744_1825".AnalogInput02;
	WeightRaw[1302].Wgt_Channel_1 AT %ID."X67AI2744_1826".AnalogInput01;
	WeightRaw[1304].Wgt_Channel_1 AT %ID."X67AI2744_1826".AnalogInput02;
	OK[1325] AT %IX."X67DM1321_1325".ModuleOk;
	OK[1327] AT %IX."X67DM1321_1327".ModuleOk;
	WeightRaw[1325].Wgt_Channel_1 AT %ID."X67AI2744_1827".AnalogInput01;
	WeightRaw[1327].Wgt_Channel_1 AT %ID."X67AI2744_1827".AnalogInput02;
	OK[1326] AT %IX."X67DM1321_1326".ModuleOk;
	OK[1328] AT %IX."X67DM1321_1328".ModuleOk;
	WeightRaw[1326].Wgt_Channel_1 AT %ID."X67AI2744_1828".AnalogInput01;
	WeightRaw[1328].Wgt_Channel_1 AT %ID."X67AI2744_1828".AnalogInput02;
	WeightRaw[1305].Wgt_Channel_1 AT %ID."X67AI2744_1829".AnalogInput01;
	WeightRaw[1307].Wgt_Channel_1 AT %ID."X67AI2744_1829".AnalogInput02;
	WeightRaw[1329].Wgt_Channel_1 AT %ID."X67AI2744_1831".AnalogInput01;
	WeightRaw[1331].Wgt_Channel_1 AT %ID."X67AI2744_1831".AnalogInput02;
	OK[1329] AT %IX."X67DM1321_1329".ModuleOk;
	OK[1331] AT %IX."X67DM1321_1331".ModuleOk;
	WeightRaw[1306].Wgt_Channel_1 AT %ID."X67AI2744_1830".AnalogInput01;
	WeightRaw[1308].Wgt_Channel_1 AT %ID."X67AI2744_1830".AnalogInput02;
	OK[1330] AT %IX."X67DM1321_1330".ModuleOk;
	OK[1332] AT %IX."X67DM1321_1332".ModuleOk;
	WeightRaw[1330].Wgt_Channel_1 AT %ID."X67AI2744_1832".AnalogInput01;
	WeightRaw[1332].Wgt_Channel_1 AT %ID."X67AI2744_1832".AnalogInput02;
	WeightRaw[1309].Wgt_Channel_1 AT %ID."X67AI2744_1833".AnalogInput01;
	WeightRaw[1311].Wgt_Channel_1 AT %ID."X67AI2744_1833".AnalogInput02;
	WeightRaw[1310].Wgt_Channel_1 AT %ID."X67AI2744_1834".AnalogInput01;
	WeightRaw[1312].Wgt_Channel_1 AT %ID."X67AI2744_1834".AnalogInput02;
	OK[1333] AT %IX."X67DM1321_1333".ModuleOk;
	OK[1335] AT %IX."X67DM1321_1335".ModuleOk;
	OK[1334] AT %IX."X67DM1321_1334".ModuleOk;
	OK[1336] AT %IX."X67DM1321_1336".ModuleOk;
	WeightRaw[1333].Wgt_Channel_1 AT %ID."X67AI2744_1835".AnalogInput01;
	WeightRaw[1335].Wgt_Channel_1 AT %ID."X67AI2744_1835".AnalogInput02;
	WeightRaw[1313].Wgt_Channel_1 AT %ID."X67AI2744_1837".AnalogInput01;
	WeightRaw[1315].Wgt_Channel_1 AT %ID."X67AI2744_1837".AnalogInput02;
	WeightRaw[1314].Wgt_Channel_1 AT %ID."X67AI2744_1838".AnalogInput01;
	WeightRaw[1316].Wgt_Channel_1 AT %ID."X67AI2744_1838".AnalogInput02;
	OK[1337] AT %IX."X67DM1321_1337".ModuleOk;
	OK[1339] AT %IX."X67DM1321_1339".ModuleOk;
	OK[1338] AT %IX."X67DM1321_1338".ModuleOk;
	OK[1340] AT %IX."X67DM1321_1340".ModuleOk;
	WeightRaw[1337].Wgt_Channel_1 AT %ID."X67AI2744_1839".AnalogInput01;
	WeightRaw[1339].Wgt_Channel_1 AT %ID."X67AI2744_1839".AnalogInput02;
	OK[1341] AT %IX."X67DM1321_1341".ModuleOk;
	OK[1343] AT %IX."X67DM1321_1343".ModuleOk;
	OK[1342] AT %IX."X67DM1321_1342".ModuleOk;
	OK[1344] AT %IX."X67DM1321_1344".ModuleOk;
	WeightRaw[1341].Wgt_Channel_1 AT %ID."X67AI2744_1843".AnalogInput01;
	WeightRaw[1343].Wgt_Channel_1 AT %ID."X67AI2744_1843".AnalogInput02;
	OK[1321] AT %IX."X67DM1321_1321".ModuleOk;
	OK[1323] AT %IX."X67DM1321_1627".ModuleOk;
	WeightRaw[1321].Wgt_Channel_1 AT %ID."X67AI2744_1845".AnalogInput01;
	WeightRaw[1323].Wgt_Channel_1 AT %ID."X67AI2744_1845".AnalogInput02;
	OK[1322] AT %IX."X67DM1321_1322".ModuleOk;
	OK[1324] AT %IX."X67DM1321_1324".ModuleOk;
	WeightRaw[1322].Wgt_Channel_1 AT %ID."X67AI2744_1846".AnalogInput01;
	WeightRaw[1324].Wgt_Channel_1 AT %ID."X67AI2744_1846".AnalogInput02;
	OK[1345] AT %IX."X67DM1321_1345".ModuleOk;
	OK[1347] AT %IX."X67DM1321_1347".ModuleOk;
	WeightRaw[1345].Wgt_Channel_1 AT %ID."X67AI2744_1847".AnalogInput01;
	WeightRaw[1347].Wgt_Channel_1 AT %ID."X67AI2744_1847".AnalogInput02;
	OK[1346] AT %IX."X67DM1321_1346".ModuleOk;
	OK[1348] AT %IX."X67DM1321_1348".ModuleOk;
	SM[1414].ModuleOk AT %IX."X67SI8103_1414".ModuleOk;
	SM[1414].ModuleID AT %IW."X67SI8103_1414".ModuleID;
	SM[1414].HardwareVariant AT %IW."X67SI8103_1414".HardwareVariant;
	SM[1414].FirmwareVersion AT %IW."X67SI8103_1414".FirmwareVersion;
	SM[1414].SafeModuleOK AT %IX."X67SI8103_1414".SafeModuleOK;
	SM[1414].SafeDigitialInput01 AT %IX."X67SI8103_1414".SafeDigitalInput01;
	SM[1414].SafeDigitialInput02 AT %IX."X67SI8103_1414".SafeDigitalInput02;
	SM[1414].SafeDigitialInput03 AT %IX."X67SI8103_1414".SafeDigitalInput03;
	SM[1414].SafeDigitialInput04 AT %IX."X67SI8103_1414".SafeDigitalInput04;
	SM[1414].SafeDigitialInput05 AT %IX."X67SI8103_1414".SafeDigitalInput05;
	SM[1414].SafeDigitialInput06 AT %IX."X67SI8103_1414".SafeDigitalInput06;
	SM[1414].SafeDigitialInput07 AT %IX."X67SI8103_1414".SafeDigitalInput07;
	SM[1414].SafeDigitialInput08 AT %IX."X67SI8103_1414".SafeDigitalInput08;
	SM[1414].SafeTwoChannelInput0102 AT %IX."X67SI8103_1414".SafeTwoChannelInput0102;
	SM[1414].SafeTwoChannelInput0304 AT %IX."X67SI8103_1414".SafeTwoChannelInput0304;
	SM[1414].SafeTwoChannelInput0506 AT %IX."X67SI8103_1414".SafeTwoChannelInput0506;
	SM[1414].SafeTwoChannelInput0708 AT %IX."X67SI8103_1414".SafeTwoChannelInput0708;
	SM[1414].DigitalInput01 AT %IX."X67SI8103_1414".DigitalInput01;
	SM[1414].DigitalInput02 AT %IX."X67SI8103_1414".DigitalInput02;
	SM[1414].DigitalOutput01 AT %QX."X67SI8103_1414".DigitalOutput01;
	SM[1414].DigitalOutput02 AT %QX."X67SI8103_1414".DigitalOutput02;
	SM[1415].ModuleOk AT %IX."X67SI8103_1415".ModuleOk;
	SM[1415].ModuleID AT %IW."X67SI8103_1415".ModuleID;
	SM[1415].HardwareVariant AT %IW."X67SI8103_1415".HardwareVariant;
	SM[1415].FirmwareVersion AT %IW."X67SI8103_1415".FirmwareVersion;
	SM[1415].SafeModuleOK AT %IX."X67SI8103_1415".SafeModuleOK;
	SM[1415].SafeDigitialInput01 AT %IX."X67SI8103_1415".SafeDigitalInput01;
	SM[1415].SafeDigitialInput02 AT %IX."X67SI8103_1415".SafeDigitalInput02;
	SM[1415].SafeDigitialInput03 AT %IX."X67SI8103_1415".SafeDigitalInput03;
	SM[1415].SafeDigitialInput04 AT %IX."X67SI8103_1415".SafeDigitalInput04;
	SM[1415].SafeDigitialInput05 AT %IX."X67SI8103_1415".SafeDigitalInput05;
	SM[1415].SafeDigitialInput06 AT %IX."X67SI8103_1415".SafeDigitalInput06;
	SM[1415].SafeDigitialInput07 AT %IX."X67SI8103_1415".SafeDigitalInput07;
	SM[1415].SafeDigitialInput08 AT %IX."X67SI8103_1415".SafeDigitalInput08;
	SM[1415].SafeTwoChannelInput0102 AT %IX."X67SI8103_1415".SafeTwoChannelInput0102;
	SM[1415].SafeTwoChannelInput0304 AT %IX."X67SI8103_1415".SafeTwoChannelInput0304;
	SM[1415].SafeTwoChannelInput0506 AT %IX."X67SI8103_1415".SafeTwoChannelInput0506;
	SM[1415].SafeTwoChannelInput0708 AT %IX."X67SI8103_1415".SafeTwoChannelInput0708;
	SM[1415].DigitalInput01 AT %IX."X67SI8103_1415".DigitalInput01;
	SM[1415].DigitalInput02 AT %IX."X67SI8103_1415".DigitalInput02;
	SM[1415].DigitalOutput01 AT %QX."X67SI8103_1415".DigitalOutput01;
	SM[1415].DigitalOutput02 AT %QX."X67SI8103_1415".DigitalOutput02;
	SM[1404].ModuleOk AT %IX."X67SI8103_1404".ModuleOk;
	SM[1404].ModuleID AT %IW."X67SI8103_1404".ModuleID;
	SM[1404].HardwareVariant AT %IW."X67SI8103_1404".HardwareVariant;
	SM[1404].FirmwareVersion AT %IW."X67SI8103_1404".FirmwareVersion;
	SM[1404].SafeModuleOK AT %IX."X67SI8103_1404".SafeModuleOK;
	SM[1404].SafeDigitialInput01 AT %IX."X67SI8103_1404".SafeDigitalInput01;
	SM[1404].SafeDigitialInput02 AT %IX."X67SI8103_1404".SafeDigitalInput02;
	SM[1404].SafeDigitialInput03 AT %IX."X67SI8103_1404".SafeDigitalInput03;
	SM[1404].SafeDigitialInput04 AT %IX."X67SI8103_1404".SafeDigitalInput04;
	SM[1404].SafeDigitialInput05 AT %IX."X67SI8103_1404".SafeDigitalInput05;
	SM[1404].SafeDigitialInput06 AT %IX."X67SI8103_1404".SafeDigitalInput06;
	SM[1404].SafeDigitialInput07 AT %IX."X67SI8103_1404".SafeDigitalInput07;
	SM[1404].SafeDigitialInput08 AT %IX."X67SI8103_1404".SafeDigitalInput08;
	SM[1404].SafeTwoChannelInput0102 AT %IX."X67SI8103_1404".SafeTwoChannelInput0102;
	SM[1404].SafeTwoChannelInput0304 AT %IX."X67SI8103_1404".SafeTwoChannelInput0304;
	SM[1404].SafeTwoChannelInput0506 AT %IX."X67SI8103_1404".SafeTwoChannelInput0506;
	SM[1404].SafeTwoChannelInput0708 AT %IX."X67SI8103_1404".SafeTwoChannelInput0708;
	SM[1404].SafeTwoChannelOk0102 AT %IX."X67SI8103_1404".SafeTwoChannelOK0102;
	SM[1404].SafeTwoChannelOk0304 AT %IX."X67SI8103_1404".SafeTwoChannelOK0304;
	SM[1404].SafeTwoChannelOk0506 AT %IX."X67SI8103_1404".SafeTwoChannelOK0506;
	SM[1404].SafeTwoChannelOk0708 AT %IX."X67SI8103_1404".SafeTwoChannelOK0708;
	SM[1404].DigitalInput01 AT %IX."X67SI8103_1404".DigitalInput01;
	SM[1404].DigitalInput02 AT %IX."X67SI8103_1404".DigitalInput02;
	SM[1404].DigitalOutput01 AT %QX."X67SI8103_1404".DigitalOutput01;
	SM[1404].DigitalOutput02 AT %QX."X67SI8103_1404".DigitalOutput02;
	SM[1409].ModuleOk AT %IX."X67SI8103_1409".ModuleOk;
	SM[1409].ModuleID AT %IW."X67SI8103_1409".ModuleID;
	SM[1409].HardwareVariant AT %IW."X67SI8103_1409".HardwareVariant;
	SM[1409].FirmwareVersion AT %IW."X67SI8103_1409".FirmwareVersion;
	SM[1409].SafeModuleOK AT %IX."X67SI8103_1409".SafeModuleOK;
	SM[1409].SafeDigitialInput01 AT %IX."X67SI8103_1409".SafeDigitalInput01;
	SM[1409].SafeDigitialInput02 AT %IX."X67SI8103_1409".SafeDigitalInput02;
	SM[1409].SafeDigitialInput03 AT %IX."X67SI8103_1409".SafeDigitalInput03;
	SM[1409].SafeDigitialInput04 AT %IX."X67SI8103_1409".SafeDigitalInput04;
	SM[1409].SafeDigitialInput05 AT %IX."X67SI8103_1409".SafeDigitalInput05;
	SM[1409].SafeDigitialInput06 AT %IX."X67SI8103_1409".SafeDigitalInput06;
	SM[1409].SafeDigitialInput07 AT %IX."X67SI8103_1409".SafeDigitalInput07;
	SM[1409].SafeDigitialInput08 AT %IX."X67SI8103_1409".SafeDigitalInput08;
	SM[1409].SafeTwoChannelInput0102 AT %IX."X67SI8103_1409".SafeTwoChannelInput0102;
	SM[1409].SafeTwoChannelInput0304 AT %IX."X67SI8103_1409".SafeTwoChannelInput0304;
	SM[1409].SafeTwoChannelInput0506 AT %IX."X67SI8103_1409".SafeTwoChannelInput0506;
	SM[1409].SafeTwoChannelInput0708 AT %IX."X67SI8103_1409".SafeTwoChannelInput0708;
	SM[1409].DigitalInput01 AT %IX."X67SI8103_1409".DigitalInput01;
	SM[1409].DigitalInput02 AT %IX."X67SI8103_1409".DigitalInput02;
	SM[1409].DigitalOutput01 AT %QX."X67SI8103_1409".DigitalOutput01;
	SM[1409].DigitalOutput02 AT %QX."X67SI8103_1409".DigitalOutput02;
	OK[1509] AT %IX."X67DM1321_1509".ModuleOk;
	SM[1408].ModuleOk AT %IX."X67SI8103_1408".ModuleOk;
	SM[1408].ModuleID AT %IW."X67SI8103_1408".ModuleID;
	SM[1408].HardwareVariant AT %IW."X67SI8103_1408".HardwareVariant;
	SM[1408].FirmwareVersion AT %IW."X67SI8103_1408".FirmwareVersion;
	SM[1408].SafeModuleOK AT %IX."X67SI8103_1408".SafeModuleOK;
	SM[1408].SafeDigitialInput01 AT %IX."X67SI8103_1408".SafeDigitalInput01;
	SM[1408].SafeDigitialInput02 AT %IX."X67SI8103_1408".SafeDigitalInput02;
	SM[1408].SafeDigitialInput03 AT %IX."X67SI8103_1408".SafeDigitalInput03;
	SM[1408].SafeDigitialInput04 AT %IX."X67SI8103_1408".SafeDigitalInput04;
	SM[1408].SafeDigitialInput05 AT %IX."X67SI8103_1408".SafeDigitalInput05;
	SM[1408].SafeDigitialInput06 AT %IX."X67SI8103_1408".SafeDigitalInput06;
	SM[1408].SafeDigitialInput07 AT %IX."X67SI8103_1408".SafeDigitalInput07;
	SM[1408].SafeDigitialInput08 AT %IX."X67SI8103_1408".SafeDigitalInput08;
	SM[1408].SafeTwoChannelInput0102 AT %IX."X67SI8103_1408".SafeTwoChannelInput0102;
	SM[1408].SafeTwoChannelInput0304 AT %IX."X67SI8103_1408".SafeTwoChannelInput0304;
	SM[1408].SafeTwoChannelInput0506 AT %IX."X67SI8103_1408".SafeTwoChannelInput0506;
	SM[1408].SafeTwoChannelInput0708 AT %IX."X67SI8103_1408".SafeTwoChannelInput0708;
	SM[1408].DigitalInput01 AT %IX."X67SI8103_1408".DigitalInput01;
	SM[1408].DigitalInput02 AT %IX."X67SI8103_1408".DigitalInput02;
	SM[1408].DigitalOutput01 AT %QX."X67SI8103_1408".DigitalOutput01;
	SM[1408].DigitalOutput02 AT %QX."X67SI8103_1408".DigitalOutput02;
	WeightRaw[1317].Wgt_Channel_1 AT %ID."X67AI2744_1841".AnalogInput01;
	WeightRaw[1319].Wgt_Channel_1 AT %ID."X67AI2744_1841".AnalogInput02;
	WeightRaw[1318].Wgt_Channel_1 AT %ID."X67AI2744_1842".AnalogInput01;
	WeightRaw[1320].Wgt_Channel_1 AT %ID."X67AI2744_1842".AnalogInput02;
	ABB_EPL.Drives[3].Comm.ModuleOk AT %IX."FEPL-02_and_ACS380_STB5".ModuleOk;
	ABB_EPL.Drives[3].Comm.ErrorCode AT %IW."FEPL-02_and_ACS380_STB5".VendorSpecificAlarmCodes_I2203;
	ABB_EPL.Drives[3].Comm.ControlWord AT %QW."FEPL-02_and_ACS380_STB5".ControlWord_I6040Out;
	ABB_EPL.Drives[3].Comm.StatusWord AT %IW."FEPL-02_and_ACS380_STB5".StatusWord_I6041;
	ABB_EPL.Drives[3].Comm.TargetVelocity AT %QW."FEPL-02_and_ACS380_STB5".VlTargetVelocity_I6042Out;
	ABB_EPL.Drives[3].Comm.ActVelocity AT %IW."FEPL-02_and_ACS380_STB5".VlVelocityActualValue_I6044;
	ABB_EPL.Drives[3].Comm.ActCurrent AT %ID."FEPL-02_and_ACS380_STB5"._0107_Motor_current_I4001_S07;
	ABB_EPL.Drives[3].Comm.ActTorque AT %ID."FEPL-02_and_ACS380_STB5"._0110_Motor_torque_I4001_S0A;
	ABB_EPL.Drives[4].Comm.ModuleOk AT %IX."FEPL-02_and_ACS380_STB6".ModuleOk;
	ABB_EPL.Drives[4].Comm.ErrorCode AT %IW."FEPL-02_and_ACS380_STB6".VendorSpecificAlarmCodes_I2203;
	ABB_EPL.Drives[4].Comm.ControlWord AT %QW."FEPL-02_and_ACS380_STB6".ControlWord_I6040Out;
	ABB_EPL.Drives[4].Comm.StatusWord AT %IW."FEPL-02_and_ACS380_STB6".StatusWord_I6041;
	ABB_EPL.Drives[4].Comm.TargetVelocity AT %QW."FEPL-02_and_ACS380_STB6".VlTargetVelocity_I6042Out;
	ABB_EPL.Drives[4].Comm.ActVelocity AT %IW."FEPL-02_and_ACS380_STB6".VlVelocityActualValue_I6044;
	ABB_EPL.Drives[4].Comm.ActCurrent AT %ID."FEPL-02_and_ACS380_STB6"._0107_Motor_current_I4001_S07;
	ABB_EPL.Drives[4].Comm.ActTorque AT %ID."FEPL-02_and_ACS380_STB6"._0110_Motor_torque_I4001_S0A;
	ABB_EPL.Drives[5].Comm.ModuleOk AT %IX."FEPL-02_and_ACS380_STB7".ModuleOk;
	ABB_EPL.Drives[5].Comm.ErrorCode AT %IW."FEPL-02_and_ACS380_STB7".VendorSpecificAlarmCodes_I2203;
	ABB_EPL.Drives[5].Comm.ControlWord AT %QW."FEPL-02_and_ACS380_STB7".ControlWord_I6040Out;
	ABB_EPL.Drives[5].Comm.StatusWord AT %IW."FEPL-02_and_ACS380_STB7".StatusWord_I6041;
	ABB_EPL.Drives[5].Comm.TargetVelocity AT %QW."FEPL-02_and_ACS380_STB7".VlTargetVelocity_I6042Out;
	ABB_EPL.Drives[5].Comm.ActVelocity AT %IW."FEPL-02_and_ACS380_STB7".VlVelocityActualValue_I6044;
	ABB_EPL.Drives[5].Comm.ActCurrent AT %ID."FEPL-02_and_ACS380_STB7"._0107_Motor_current_I4001_S07;
	ABB_EPL.Drives[5].Comm.ActTorque AT %ID."FEPL-02_and_ACS380_STB7"._0110_Motor_torque_I4001_S0A;
	ABB_EPL.Drives[6].Comm.ModuleOk AT %IX."FEPL-02_and_ACS380_STB3".ModuleOk;
	ABB_EPL.Drives[6].Comm.ErrorCode AT %IW."FEPL-02_and_ACS380_STB3".VendorSpecificAlarmCodes_I2203;
	ABB_EPL.Drives[6].Comm.ControlWord AT %QW."FEPL-02_and_ACS380_STB3".ControlWord_I6040Out;
	ABB_EPL.Drives[6].Comm.StatusWord AT %IW."FEPL-02_and_ACS380_STB3".StatusWord_I6041;
	ABB_EPL.Drives[6].Comm.TargetVelocity AT %QW."FEPL-02_and_ACS380_STB3".VlTargetVelocity_I6042Out;
	ABB_EPL.Drives[6].Comm.ActVelocity AT %IW."FEPL-02_and_ACS380_STB3".VlVelocityActualValue_I6044;
	ABB_EPL.Drives[6].Comm.ActCurrent AT %ID."FEPL-02_and_ACS380_STB3"._0107_Motor_current_I4001_S07;
	ABB_EPL.Drives[6].Comm.ActTorque AT %ID."FEPL-02_and_ACS380_STB3"._0110_Motor_torque_I4001_S0A;
	ABB_EPL.Drives[7].Comm.ModuleOk AT %IX."FEPL-02_and_ACS380_STB4".ModuleOk;
	ABB_EPL.Drives[7].Comm.ErrorCode AT %IW."FEPL-02_and_ACS380_STB4".VendorSpecificAlarmCodes_I2203;
	ABB_EPL.Drives[7].Comm.ControlWord AT %QW."FEPL-02_and_ACS380_STB4".ControlWord_I6040Out;
	ABB_EPL.Drives[7].Comm.StatusWord AT %IW."FEPL-02_and_ACS380_STB4".StatusWord_I6041;
	ABB_EPL.Drives[7].Comm.TargetVelocity AT %QW."FEPL-02_and_ACS380_STB4".VlTargetVelocity_I6042Out;
	ABB_EPL.Drives[7].Comm.ActVelocity AT %IW."FEPL-02_and_ACS380_STB4".VlVelocityActualValue_I6044;
	ABB_EPL.Drives[7].Comm.ActCurrent AT %ID."FEPL-02_and_ACS380_STB4"._0107_Motor_current_I4001_S07;
	ABB_EPL.Drives[7].Comm.ActTorque AT %ID."FEPL-02_and_ACS380_STB4"._0110_Motor_torque_I4001_S0A;
	ABB_EPL.Drives[8].Comm.ModuleOk AT %IX."FEPL-02_and_ACS380_STB8".ModuleOk;
	ABB_EPL.Drives[8].Comm.ErrorCode AT %IW."FEPL-02_and_ACS380_STB8".VendorSpecificAlarmCodes_I2203;
	ABB_EPL.Drives[8].Comm.ControlWord AT %QW."FEPL-02_and_ACS380_STB8".ControlWord_I6040Out;
	ABB_EPL.Drives[8].Comm.StatusWord AT %IW."FEPL-02_and_ACS380_STB8".StatusWord_I6041;
	ABB_EPL.Drives[8].Comm.TargetVelocity AT %QW."FEPL-02_and_ACS380_STB8".VlTargetVelocity_I6042Out;
	ABB_EPL.Drives[8].Comm.ActVelocity AT %IW."FEPL-02_and_ACS380_STB8".VlVelocityActualValue_I6044;
	ABB_EPL.Drives[8].Comm.ActCurrent AT %ID."FEPL-02_and_ACS380_STB8"._0107_Motor_current_I4001_S07;
	ABB_EPL.Drives[8].Comm.ActTorque AT %ID."FEPL-02_and_ACS380_STB8"._0110_Motor_torque_I4001_S0A;
	ABB_EPL.Drives[9].Comm.ModuleOk AT %IX."FEPL-02_and_ACS380_STB9".ModuleOk;
	ABB_EPL.Drives[9].Comm.ErrorCode AT %IW."FEPL-02_and_ACS380_STB9".VendorSpecificAlarmCodes_I2203;
	ABB_EPL.Drives[9].Comm.ControlWord AT %QW."FEPL-02_and_ACS380_STB9".ControlWord_I6040Out;
	ABB_EPL.Drives[9].Comm.StatusWord AT %IW."FEPL-02_and_ACS380_STB9".StatusWord_I6041;
	ABB_EPL.Drives[9].Comm.TargetVelocity AT %QW."FEPL-02_and_ACS380_STB9".VlTargetVelocity_I6042Out;
	ABB_EPL.Drives[9].Comm.ActVelocity AT %IW."FEPL-02_and_ACS380_STB9".VlVelocityActualValue_I6044;
	ABB_EPL.Drives[9].Comm.ActCurrent AT %ID."FEPL-02_and_ACS380_STB9"._0107_Motor_current_I4001_S07;
	ABB_EPL.Drives[9].Comm.ActTorque AT %ID."FEPL-02_and_ACS380_STB9"._0110_Motor_torque_I4001_S0A;
	ABB_EPL.Drives[10].Comm.ModuleOk AT %IX."FEPL-02_and_ACS380_STB10".ModuleOk;
	ABB_EPL.Drives[10].Comm.ErrorCode AT %IW."FEPL-02_and_ACS380_STB10".VendorSpecificAlarmCodes_I2203;
	ABB_EPL.Drives[10].Comm.ControlWord AT %QW."FEPL-02_and_ACS380_STB10".ControlWord_I6040Out;
	ABB_EPL.Drives[10].Comm.StatusWord AT %IW."FEPL-02_and_ACS380_STB10".StatusWord_I6041;
	ABB_EPL.Drives[10].Comm.TargetVelocity AT %QW."FEPL-02_and_ACS380_STB10".VlTargetVelocity_I6042Out;
	ABB_EPL.Drives[10].Comm.ActVelocity AT %IW."FEPL-02_and_ACS380_STB10".VlVelocityActualValue_I6044;
	ABB_EPL.Drives[10].Comm.ActCurrent AT %ID."FEPL-02_and_ACS380_STB10"._0107_Motor_current_I4001_S07;
	ABB_EPL.Drives[10].Comm.ActTorque AT %ID."FEPL-02_and_ACS380_STB10"._0110_Motor_torque_I4001_S0A;
	ABB_EPL.Drives[13].Comm.ModuleOk AT %IX."FEPL-02_and_ACS380_SB3".ModuleOk;
	ABB_EPL.Drives[13].Comm.ErrorCode AT %IW."FEPL-02_and_ACS380_SB3".VendorSpecificAlarmCodes_I2203;
	ABB_EPL.Drives[13].Comm.ControlWord AT %QW."FEPL-02_and_ACS380_SB3".ControlWord_I6040Out;
	ABB_EPL.Drives[13].Comm.StatusWord AT %IW."FEPL-02_and_ACS380_SB3".StatusWord_I6041;
	ABB_EPL.Drives[13].Comm.TargetVelocity AT %QW."FEPL-02_and_ACS380_SB3".VlTargetVelocity_I6042Out;
	ABB_EPL.Drives[13].Comm.ActVelocity AT %IW."FEPL-02_and_ACS380_SB3".VlVelocityActualValue_I6044;
	ABB_EPL.Drives[13].Comm.ActCurrent AT %ID."FEPL-02_and_ACS380_SB3"._0107_Motor_current_I4001_S07;
	ABB_EPL.Drives[13].Comm.ActTorque AT %ID."FEPL-02_and_ACS380_SB3"._0110_Motor_torque_I4001_S0A;
	ABB_EPL.Drives[14].Comm.ModuleOk AT %IX."FEPL-02_and_ACS380_SB4".ModuleOk;
	ABB_EPL.Drives[14].Comm.ErrorCode AT %IW."FEPL-02_and_ACS380_SB4".VendorSpecificAlarmCodes_I2203;
	ABB_EPL.Drives[14].Comm.ControlWord AT %QW."FEPL-02_and_ACS380_SB4".ControlWord_I6040Out;
	ABB_EPL.Drives[14].Comm.StatusWord AT %IW."FEPL-02_and_ACS380_SB4".StatusWord_I6041;
	ABB_EPL.Drives[14].Comm.TargetVelocity AT %QW."FEPL-02_and_ACS380_SB4".VlTargetVelocity_I6042Out;
	ABB_EPL.Drives[14].Comm.ActVelocity AT %IW."FEPL-02_and_ACS380_SB4".VlVelocityActualValue_I6044;
	ABB_EPL.Drives[14].Comm.ActCurrent AT %ID."FEPL-02_and_ACS380_SB4"._0107_Motor_current_I4001_S07;
	ABB_EPL.Drives[14].Comm.ActTorque AT %ID."FEPL-02_and_ACS380_SB4"._0110_Motor_torque_I4001_S0A;
	ABB_EPL.Drives[15].Comm.ModuleOk AT %IX."FEPL-02_and_ACS380_STB11".ModuleOk;
	ABB_EPL.Drives[15].Comm.ErrorCode AT %IW."FEPL-02_and_ACS380_STB11".VendorSpecificAlarmCodes_I2203;
	ABB_EPL.Drives[15].Comm.ControlWord AT %QW."FEPL-02_and_ACS380_STB11".ControlWord_I6040Out;
	ABB_EPL.Drives[15].Comm.StatusWord AT %IW."FEPL-02_and_ACS380_STB11".StatusWord_I6041;
	ABB_EPL.Drives[15].Comm.TargetVelocity AT %QW."FEPL-02_and_ACS380_STB11".VlTargetVelocity_I6042Out;
	ABB_EPL.Drives[15].Comm.ActVelocity AT %IW."FEPL-02_and_ACS380_STB11".VlVelocityActualValue_I6044;
	ABB_EPL.Drives[15].Comm.ActCurrent AT %ID."FEPL-02_and_ACS380_STB11"._0107_Motor_current_I4001_S07;
	ABB_EPL.Drives[15].Comm.ActTorque AT %ID."FEPL-02_and_ACS380_STB11"._0110_Motor_torque_I4001_S0A;
	ABB_EPL.Drives[16].Comm.ModuleOk AT %IX."FEPL-02_and_ACS380_STB12".ModuleOk;
	ABB_EPL.Drives[16].Comm.ErrorCode AT %IW."FEPL-02_and_ACS380_STB12".VendorSpecificAlarmCodes_I2203;
	ABB_EPL.Drives[16].Comm.ControlWord AT %QW."FEPL-02_and_ACS380_STB12".ControlWord_I6040Out;
	ABB_EPL.Drives[16].Comm.StatusWord AT %IW."FEPL-02_and_ACS380_STB12".StatusWord_I6041;
	ABB_EPL.Drives[16].Comm.TargetVelocity AT %QW."FEPL-02_and_ACS380_STB12".VlTargetVelocity_I6042Out;
	ABB_EPL.Drives[16].Comm.ActVelocity AT %IW."FEPL-02_and_ACS380_STB12".VlVelocityActualValue_I6044;
	ABB_EPL.Drives[16].Comm.ActCurrent AT %ID."FEPL-02_and_ACS380_STB12"._0107_Motor_current_I4001_S07;
	ABB_EPL.Drives[16].Comm.ActTorque AT %ID."FEPL-02_and_ACS380_STB12"._0110_Motor_torque_I4001_S0A;
END_VAR
```

### addmoduleOk.rb - APC2200/addmoduleOk.rb
```
dirname = Dir.pwd
fileName = dirname + '/iomap.iom'
modules = Array.new
exclusionList = Array.new

file = File.open(fileName)
file.each do |line|
  if line.include? "X["
    pos1 = line.index("X[") + 2
    pos2 = line.index("].X") - 1
    number = line[pos1..pos2]
    pos1 = line.index("%IX.") + 4
    pos2 = line.index(".DigitalInput") - 1
    name = line[pos1..pos2]
    modules << [number,name]
  elsif line.include? "Y["
    pos1 = line.index("Y[") + 2
    pos2 = line.index("].Y") - 1
    number = line[pos1..pos2]
    pos1 = line.index("%QX.") + 4
    pos2 = line.index(".DigitalOutput") - 1
    name = line[pos1..pos2]
    modules << [number,name]
  end
end

#-- Read through the file again to see if we have already written the OK.
file = File.open(fileName)
file.each do |line|
  if line.include? "OK["
    pos1 = line.index("OK[") + 3
    pos2 = line.index("] AT") - 1
    number = line[pos1..pos2]
    exclusionList << number
  end
end

writecount = 0
excludecount = 0
wd = ""

modules.uniq.each do |x|
  unless exclusionList.uniq.include?x[0]
   #puts "will write #{x[0]} -- #{x[1]}"
    writecount += 1
    wd << "\tOK[#{x[0]}] AT %IX.#{x[1]}.ModuleOk;\n"
  else
    #puts "already in list #{x[0]} "
    excludecount += 1
  end
end
wd << "END_VAR\n"

file = File.read(fileName)
file.gsub!("END_VAR\n","")

file << wd
#puts file
fo = File.open(fileName,"w")
fo.write(file)
fo.close
puts "added #{writecount} modules, found #{excludecount} existing "
```

### Config.mpaudittrail - APC2200/mappServices/Config.mpaudittrail
```
Element gAuditTrail (Type=mpaudittrail)
  Audit:
    Events:
      [0] = 16
      [1]
      [2]
    TextSource:
      OutputFormat = Value of [%dpid] changed. Old: [%old$12.0], New: [%new$12.0]
    Export:
      Encrypt = FALSE
  Monitor:
    0:
      pv = BusCouplerDiag[21].ModuleLostWhilstOperational
    1:
      pv = BusCouplerDiag[21].StationAtBusEnd
    2:
      pv = BusCouplerDiag[21].StationPastInFrameError
    3:
      pv = BusCouplerDiag[21].StationPastOutFrameError
    4:
      pv = BusCouplerDiag[22].ModuleLostWhilstOperational
    5:
      pv = BusCouplerDiag[22].StationAtBusEnd
    6:
      pv = BusCouplerDiag[22].StationPastInFrameError
    7:
      pv = BusCouplerDiag[22].StationPastOutFrameError
    8:
      pv = BusCouplerDiag[31].ModuleLostWhilstOperational
    9:
      pv = BusCouplerDiag[31].StationAtBusEnd
    10:
      pv = BusCouplerDiag[31].StationPastInFrameError
    11:
      pv = BusCouplerDiag[31].StationPastOutFrameError
    12:
      pv = BusCouplerDiag[32].ModuleLostWhilstOperational
    13:
      pv = BusCouplerDiag[32].StationAtBusEnd
    14:
      pv = BusCouplerDiag[32].StationPastInFrameError
    15:
      pv = BusCouplerDiag[32].StationPastOutFrameError
    16:
      pv = BusCouplerDiag[33].ModuleLostWhilstOperational
    17:
      pv = BusCouplerDiag[33].StationAtBusEnd
    18:
      pv = BusCouplerDiag[33].StationPastInFrameError
    19:
      pv = BusCouplerDiag[33].StationPastOutFrameError
    20:
      pv = BusCouplerDiag[34].ModuleLostWhilstOperational
    21:
      pv = BusCouplerDiag[34].StationAtBusEnd
    22:
      pv = BusCouplerDiag[34].StationPastInFrameError
    23:
      pv = BusCouplerDiag[34].StationPastOutFrameError
    24:
      pv = BusCouplerDiag[35].ModuleLostWhilstOperational
    25:
      pv = BusCouplerDiag[35].StationAtBusEnd
    26:
      pv = BusCouplerDiag[35].StationPastInFrameError
    27:
      pv = BusCouplerDiag[35].StationPastOutFrameError
    28:
      pv = BusCouplerDiag[41].ModuleLostWhilstOperational
    29:
      pv = BusCouplerDiag[41].StationAtBusEnd
    30:
      pv = BusCouplerDiag[41].StationPastInFrameError
    31:
      pv = BusCouplerDiag[41].StationPastOutFrameError
    32:
      pv = BusCouplerDiag[42].ModuleLostWhilstOperational
    33:
      pv = BusCouplerDiag[42].StationAtBusEnd
    34:
      pv = BusCouplerDiag[42].StationPastInFrameError
    35:
      pv = BusCouplerDiag[42].StationPastOutFrameError
    36:
      pv = BusCouplerDiag[43].ModuleLostWhilstOperational
    37:
      pv = BusCouplerDiag[43].StationAtBusEnd
    38:
      pv = BusCouplerDiag[43].StationPastInFrameError
    39:
      pv = BusCouplerDiag[43].StationPastOutFrameError
    40:
      pv = BusCouplerDiag[44].ModuleLostWhilstOperational
    41:
      pv = BusCouplerDiag[44].StationAtBusEnd
    42:
      pv = BusCouplerDiag[44].StationPastInFrameError
    43:
      pv = BusCouplerDiag[44].StationPastOutFrameError
    44:
      pv = BusCouplerDiag[45].ModuleLostWhilstOperational
    45:
      pv = BusCouplerDiag[45].StationAtBusEnd
    46:
      pv = BusCouplerDiag[45].StationPastInFrameError
    47:
      pv = BusCouplerDiag[45].StationPastOutFrameError
    48:
      pv = BusCouplerDiag[110].ModuleLostWhilstOperational
    49:
      pv = BusCouplerDiag[110].StationAtBusEnd
    50:
      pv = BusCouplerDiag[110].StationPastInFrameError
    51:
      pv = BusCouplerDiag[110].StationPastOutFrameError
```

### Settings.vicfg - APC2200/mappVision/Settings.vicfg
```
Element VisionSettings (Type=vicfg)
  ActivateVisualization = FALSE
  FileDeviceName
  Permissions:
    WriteAccessRole = Administrators
```

### viComp.visioncomponent - APC2200/mappVision/viComp.visioncomponent
```
Element gCamera_2 (Type=visioncomponent)
  VisionApplicationReference = ViAppBarcode
Element gCamera_1 (Type=visioncomponent)
  VisionApplicationReference = ViAppBarcode
Element gCamera_3 (Type=visioncomponent)
  VisionApplicationReference = ViAppBarcode
Element gCamera_4 (Type=visioncomponent)
  VisionApplicationReference = ViAppBarcode
Element gCamera_5 (Type=visioncomponent)
  VisionApplicationReference = ViAppBarcode
```

## Logical view

Binary libraries used (declarations not repeated): AsEPL, AsOpcUac, DataObj, AsXml, CAN_Lib, AsARCfg, runtime, AsBrMath, AsIecCon, astime, asstring, operator, standard, AsBrStr, AsTCP, FileIO, sys_lib, AsUDP, brsystem, ArSsl, ArUser, AsZip, powerlnk, AsETH, AsIODiag, AsHttp, AsIOAcc, AsIoTrc, AsIOLink, AsIO, MpServer, ViBase, MTBasics, MTTypes, MpAudit, MpBase, SfDomain 5.15.0, AsBrWStr, ETHERNET, AsArLog, AsUSB, AsMem, AsDb, AsFifo, AsCANopen

### Global.var - Global variables
```iecst
VAR CONSTANT
	RAIL_COUNT : UINT := 74; (**GENERATED VALUE FOR ACTUAL NUMBER OF RAILS*)
	SLING_INPUTS_COUNT : UINT := 0; (**GENERATED VALUE FOR ACTUAL NUMBER OF SLING INPUT STATIONS*)
END_VAR
VAR
	eVueServerIP : STRING[20] := '10.8.15.119';
	RailComm : ARRAY[0..RAIL_COUNT] OF RailComm_typ;
	SlingInputComm : ARRAY[0..SLING_INPUTS_COUNT] OF SlingInput_typ;
	X : ARRAY[0..3000] OF bnr_io;
	Y : ARRAY[0..3000] OF bnr_io;
	OK : ARRAY[0..3000] OF BOOL;
	spare : BOOL;
	SPARE : BOOL;
	spare_input : BOOL;
	spare_output : BOOL;
	unknown_input : BOOL;
	unknown_output : BOOL;
	mbSlaveStep : INT := 0;
	plc_info1 : WORD;
	plc_info2 : WORD;
	plc_info3 : WORD;
	plc_info4 : WORD;
	plc_info5 : WORD;
	plc_info6 : WORD;
	plc_info7 : WORD;
	plc_info8 : WORD;
	plc_info9 : WORD;
	plc_info10 : WORD;
	plc_info11 : WORD;
	plc_info12 : WORD;
	plc_info13 : WORD;
	plc_info14 : WORD;
	plc_info15 : WORD;
	plc_info16 : WORD;
	plc_info17 : WORD;
	plc_info18 : WORD;
	plc_info19 : WORD;
	plc_info20 : WORD;
	soiled_max_weight : UINT;
	clean_max_weight : UINT;
	customer_bag_max_weight : UINT;
	commArray1 : ARRAY[0..4001] OF WORD;
	commArray2 : ARRAY[0..4001] OF WORD;
	commArray3 : ARRAY[0..4001] OF WORD;
	commArray4 : ARRAY[0..4001] OF WORD;
	ss1 : BOOL;
	ss2 : BOOL;
	ss3 : BOOL;
	ss4 : BOOL;
	ss5 : BOOL;
	ss6 : BOOL;
	ss7 : BOOL;
	ss8 : BOOL;
	ss9 : BOOL;
	ss10 : BOOL;
	ss1_prs : BOOL;
	ss2_prs : BOOL;
	ss3_prs : BOOL;
	ss4_prs : BOOL;
	ss5_prs : BOOL;
	ss6_prs : BOOL;
	ss7_prs : BOOL;
	ss8_prs : BOOL;
	ss9_prs : BOOL;
	ss10_prs : BOOL;
	rail_udp_array : ARRAY[1..74] OF RailUdpType;
	r1 : rail;
	r2 : rail;
	r3 : rail;
	r4 : rail;
	r5 : rail;
	r6 : rail;
	r7 : rail;
	r8 : rail;
	r9 : rail;
	r10 : rail;
	r11 : rail;
	r12 : rail;
	r13 : rail;
	r14 : rail;
	r15 : rail;
	r16 : rail;
	r17 : rail;
	r18 : rail;
	r19 : rail;
	r20 : rail;
	r21 : rail;
	r22 : rail;
	r23 : rail;
	r24 : rail;
	r25 : rail;
	r26 : rail;
	r27 : rail;
	r28 : rail;
	r29 : rail;
	r30 : rail;
	r31 : rail;
	r32 : rail;
	r33 : rail;
	r34 : rail;
	r35 : rail;
	r36 : rail;
	r37 : rail;
	r38 : rail;
	r39 : rail;
	r40 : rail;
	r41 : rail;
	r42 : rail;
	r43 : rail;
	r44 : rail;
	r45 : rail;
	r46 : rail;
	r47 : rail;
	r48 : rail;
	r49 : rail;
	r50 : rail;
	r51 : rail;
	r52 : rail;
	r53 : rail;
	r54 : rail;
	r55 : rail;
	r56 : rail;
	r57 : rail;
	r58 : rail;
	r59 : rail;
	r60 : rail;
	r61 : rail;
	r61_R_TRIG : R_TRIG;
	r61_F_TRIG : F_TRIG;
	r62 : rail;
	r62_R_TRIG : R_TRIG;
	r62_F_TRIG : F_TRIG;
	r63 : rail;
	r63_R_TRIG : R_TRIG;
	r63_F_TRIG : F_TRIG;
	r64 : rail;
	r64_R_TRIG : R_TRIG;
	r64_F_TRIG : F_TRIG;
	r65 : rail;
	r65_R_TRIG : R_TRIG;
	r65_F_TRIG : F_TRIG;
	r66 : rail;
	r66_R_TRIG : R_TRIG;
	r66_F_TRIG : F_TRIG;
	r67 : rail;
	r67_R_TRIG : R_TRIG;
	r67_F_TRIG : F_TRIG;
	r68 : rail;
	r68_R_TRIG : R_TRIG;
	r68_F_TRIG : F_TRIG;
	r69 : rail;
	r69_R_TRIG : R_TRIG;
	r69_F_TRIG : F_TRIG;
	r70 : rail;
	r70_R_TRIG : R_TRIG;
	r70_F_TRIG : F_TRIG;
	r71 : rail;
	r72 : rail;
	r73 : rail;
	r74 : rail;
	one_sec_pulse : TON;
	not_one_sec_pulse : TON;
	thirty_msec_pulse : TON;
	not_thirty_msec_pulse : TON;
	ip : STRING;
	StartStop : BOOL;
	WeightRaw : ARRAY[1300..1620] OF Weight_typ;
	validation_alarm : BOOL;
	halted : BOOL;
	server_status : WORD;
	system_alarm_1 : BOOL;
	strobe1 : BOOL;
	horn1 : BOOL;
	soiled_validation_alarm : BOOL;
	system_alarm_2 : BOOL;
	strobe2 : BOOL;
	horn2 : BOOL;
	clean_validation_alarm : BOOL;
	rail_alarm_time_1 : INT;
	rail_signal_1 : WORD;
	rail_status_1 : WORD;
	rail_state_1 : UINT;
	rail_alarm_time_2 : INT;
	rail_signal_2 : WORD;
	rail_status_2 : WORD;
	rail_state_2 : UINT;
	rail_alarm_time_3 : INT;
	rail_signal_3 : WORD;
	rail_status_3 : WORD;
	rail_state_3 : UINT;
	rail_alarm_time_4 : INT;
	rail_signal_4 : WORD;
	rail_status_4 : WORD;
	rail_state_4 : UINT;
	rail_alarm_time_5 : INT;
	rail_signal_5 : WORD;
	rail_status_5 : WORD;
	rail_state_5 : UINT;
	rail_alarm_time_6 : INT;
	rail_signal_6 : WORD;
	rail_status_6 : WORD;
	rail_state_6 : UINT;
	rail_alarm_time_7 : INT;
	rail_signal_7 : WORD;
	rail_status_7 : WORD;
	rail_state_7 : UINT;
	rail_alarm_time_8 : INT;
	rail_signal_8 : WORD;
	rail_status_8 : WORD;
	rail_state_8 : UINT;
	rail_alarm_time_9 : INT;
	rail_signal_9 : WORD;
	rail_status_9 : WORD;
	rail_state_9 : UINT;
	rail_alarm_time_10 : INT;
	rail_signal_10 : WORD;
	rail_status_10 : WORD;
	rail_state_10 : UINT;
	rail_alarm_time_11 : INT;
	rail_signal_11 : WORD;
	rail_status_11 : WORD;
	rail_state_11 : UINT;
	rail_alarm_time_12 : INT;
	rail_signal_12 : WORD;
	rail_status_12 : WORD;
	rail_state_12 : UINT;
	rail_alarm_time_13 : INT;
	rail_signal_13 : WORD;
	rail_status_13 : WORD;
	rail_state_13 : UINT;
	rail_alarm_time_14 : INT;
	rail_signal_14 : WORD;
	rail_status_14 : WORD;
	rail_state_14 : UINT;
	rail_alarm_time_15 : INT;
	rail_signal_15 : WORD;
	rail_status_15 : WORD;
	rail_state_15 : UINT;
	rail_alarm_time_16 : INT;
	rail_signal_16 : WORD;
	rail_status_16 : WORD;
	rail_state_16 : UINT;
	rail_alarm_time_17 : INT;
	rail_signal_17 : WORD;
	rail_status_17 : WORD;
	rail_state_17 : UINT;
	rail_alarm_time_18 : INT;
	rail_signal_18 : WORD;
	rail_status_18 : WORD;
	rail_state_18 : UINT;
	rail_alarm_time_19 : INT;
	rail_signal_19 : WORD;
	rail_status_19 : WORD;
	rail_state_19 : UINT;
	rail_alarm_time_20 : INT;
	rail_signal_20 : WORD;
	rail_status_20 : WORD;
	rail_state_20 : UINT;
	rail_alarm_time_21 : INT;
	rail_signal_21 : WORD;
	rail_status_21 : WORD;
	rail_state_21 : UINT;
	rail_alarm_time_22 : INT;
	rail_signal_22 : WORD;
	rail_status_22 : WORD;
	rail_state_22 : UINT;
	rail_alarm_time_23 : INT;
	rail_signal_23 : WORD;
	rail_status_23 : WORD;
	rail_state_23 : UINT;
	rail_alarm_time_24 : INT;
	rail_signal_24 : WORD;
	rail_status_24 : WORD;
	rail_state_24 : UINT;
	rail_alarm_time_25 : INT;
	rail_signal_25 : WORD;
	rail_status_25 : WORD;
	rail_state_25 : UINT;
	rail_alarm_time_26 : INT;
	rail_signal_26 : WORD;
	rail_status_26 : WORD;
	rail_state_26 : UINT;
	rail_alarm_time_27 : INT;
	rail_signal_27 : WORD;
	rail_status_27 : WORD;
	rail_state_27 : UINT;
	rail_alarm_time_28 : INT;
	rail_signal_28 : WORD;
	rail_status_28 : WORD;
	rail_state_28 : UINT;
	rail_alarm_time_29 : INT;
	rail_signal_29 : WORD;
	rail_status_29 : WORD;
	rail_state_29 : UINT;
	rail_alarm_time_30 : INT;
	rail_signal_30 : WORD;
	rail_status_30 : WORD;
	rail_state_30 : UINT;
	rail_alarm_time_31 : INT;
	rail_signal_31 : WORD;
	rail_status_31 : WORD;
	rail_state_31 : UINT;
	rail_alarm_time_32 : INT;
	rail_signal_32 : WORD;
	rail_status_32 : WORD;
	rail_state_32 : UINT;
	rail_alarm_time_33 : INT;
	rail_signal_33 : WORD;
	rail_status_33 : WORD;
	rail_state_33 : UINT;
	rail_alarm_time_34 : INT;
	rail_signal_34 : WORD;
	rail_status_34 : WORD;
	rail_state_34 : UINT;
	rail_alarm_time_35 : INT;
	rail_signal_35 : WORD;
	rail_status_35 : WORD;
	rail_state_35 : UINT;
	rail_alarm_time_36 : INT;
	rail_signal_36 : WORD;
	rail_status_36 : WORD;
	rail_state_36 : UINT;
	rail_alarm_time_37 : INT;
	rail_signal_37 : WORD;
	rail_status_37 : WORD;
	rail_state_37 : UINT;
	rail_alarm_time_38 : INT;
	rail_signal_38 : WORD;
	rail_status_38 : WORD;
	rail_state_38 : UINT;
	rail_alarm_time_39 : INT;
	rail_signal_39 : WORD;
	rail_status_39 : WORD;
	rail_state_39 : UINT;
	rail_alarm_time_40 : INT;
	rail_signal_40 : WORD;
	rail_status_40 : WORD;
	rail_state_40 : UINT;
	rail_alarm_time_41 : INT;
	rail_signal_41 : WORD;
	rail_status_41 : WORD;
	rail_state_41 : UINT;
	rail_alarm_time_42 : INT;
	rail_signal_42 : WORD;
	rail_status_42 : WORD;
	rail_state_42 : UINT;
	rail_alarm_time_43 : INT;
	rail_signal_43 : WORD;
	rail_status_43 : WORD;
	rail_state_43 : UINT;
	rail_alarm_time_44 : INT;
	rail_signal_44 : WORD;
	rail_status_44 : WORD;
	rail_state_44 : UINT;
	rail_alarm_time_45 : INT;
	rail_signal_45 : WORD;
	rail_status_45 : WORD;
	rail_state_45 : UINT;
	rail_alarm_time_46 : INT;
	rail_signal_46 : WORD;
	rail_status_46 : WORD;
	rail_state_46 : UINT;
	rail_alarm_time_47 : INT;
	rail_signal_47 : WORD;
	rail_status_47 : WORD;
	rail_state_47 : UINT;
	rail_alarm_time_48 : INT;
	rail_signal_48 : WORD;
	rail_status_48 : WORD;
	rail_state_48 : UINT;
	rail_alarm_time_49 : INT;
	rail_signal_49 : WORD;
	rail_status_49 : WORD;
	rail_state_49 : UINT;
	rail_alarm_time_50 : INT;
	rail_signal_50 : WORD;
	rail_status_50 : WORD;
	rail_state_50 : UINT;
	rail_alarm_time_51 : INT;
	rail_signal_51 : WORD;
	rail_status_51 : WORD;
	rail_state_51 : UINT;
	rail_alarm_time_52 : INT;
	rail_signal_52 : WORD;
	rail_status_52 : WORD;
	rail_state_52 : UINT;
	rail_alarm_time_53 : INT;
	rail_signal_53 : WORD;
	rail_status_53 : WORD;
	rail_state_53 : UINT;
	rail_alarm_time_54 : INT;
	rail_signal_54 : WORD;
	rail_status_54 : WORD;
	rail_state_54 : UINT;
	rail_alarm_time_55 : INT;
	rail_signal_55 : WORD;
	rail_status_55 : WORD;
	rail_state_55 : UINT;
	rail_alarm_time_56 : INT;
	rail_signal_56 : WORD;
	rail_status_56 : WORD;
	rail_state_56 : UINT;
	rail_alarm_time_57 : INT;
	rail_signal_57 : WORD;
	rail_status_57 : WORD;
	rail_state_57 : UINT;
	rail_alarm_time_58 : INT;
	rail_signal_58 : WORD;
	rail_status_58 : WORD;
	rail_state_58 : UINT;
	rail_alarm_time_59 : INT;
	rail_signal_59 : WORD;
	rail_status_59 : WORD;
	rail_state_59 : UINT;
	rail_alarm_time_60 : INT;
	rail_signal_60 : WORD;
	rail_status_60 : WORD;
	rail_state_60 : UINT;
	rail_alarm_time_61 : INT;
	rail_signal_61 : WORD;
	rail_status_61 : WORD;
	rail_state_61 : UINT;
	rail_alarm_time_62 : INT;
	rail_signal_62 : WORD;
	rail_status_62 : WORD;
	rail_state_62 : UINT;
	rail_alarm_time_63 : INT;
	rail_signal_63 : WORD;
	rail_status_63 : WORD;
	rail_state_63 : UINT;
	rail_alarm_time_64 : INT;
	rail_signal_64 : WORD;
	rail_status_64 : WORD;
	rail_state_64 : UINT;
	rail_alarm_time_65 : INT;
	rail_signal_65 : WORD;
	rail_status_65 : WORD;
	rail_state_65 : UINT;
	rail_alarm_time_66 : INT;
	rail_signal_66 : WORD;
	rail_status_66 : WORD;
	rail_state_66 : UINT;
	rail_alarm_time_67 : INT;
	rail_signal_67 : WORD;
	rail_status_67 : WORD;
	rail_state_67 : UINT;
	rail_alarm_time_68 : INT;
	rail_signal_68 : WORD;
	rail_status_68 : WORD;
	rail_state_68 : UINT;
	rail_alarm_time_69 : INT;
	rail_signal_69 : WORD;
	rail_status_69 : WORD;
	rail_state_69 : UINT;
	rail_alarm_time_70 : INT;
	rail_signal_70 : WORD;
	rail_status_70 : WORD;
	rail_state_70 : UINT;
	rail_alarm_time_71 : INT;
	rail_signal_71 : WORD;
	rail_status_71 : WORD;
	rail_state_71 : UINT;
	rail_alarm_time_72 : INT;
	rail_signal_72 : WORD;
	rail_status_72 : WORD;
	rail_state_72 : UINT;
	rail_alarm_time_73 : INT;
	rail_signal_73 : WORD;
	rail_status_73 : WORD;
	rail_state_73 : UINT;
	rail_alarm_time_74 : INT;
	rail_signal_74 : WORD;
	rail_status_74 : WORD;
	rail_state_74 : UINT;
	conveyor_module_1_value_1 : INT;
	conveyor_module_1_value_2 : INT;
	conveyor_module_1_value_3 : INT;
	conveyor_module_1_value_4 : INT;
	conveyor_module_2_value_1 : INT;
	conveyor_module_2_value_2 : INT;
	conveyor_module_2_value_3 : INT;
	conveyor_module_2_value_4 : INT;
	conveyor_module_3_value_1 : INT;
	conveyor_module_3_value_2 : INT;
	conveyor_module_3_value_3 : INT;
	conveyor_module_3_value_4 : INT;
	conveyor_module_4_value_1 : INT;
	conveyor_module_4_value_2 : INT;
	conveyor_module_4_value_3 : INT;
	conveyor_module_4_value_4 : INT;
	conveyor_module_5_value_1 : INT;
	conveyor_module_5_value_2 : INT;
	conveyor_module_5_value_3 : INT;
	conveyor_module_5_value_4 : INT;
	conveyor_module_6_value_1 : INT;
	conveyor_module_6_value_2 : INT;
	conveyor_module_6_value_3 : INT;
	conveyor_module_6_value_4 : INT;
	conveyor_module_7_value_1 : INT;
	conveyor_module_7_value_2 : INT;
	conveyor_module_7_value_3 : INT;
	conveyor_module_7_value_4 : INT;
	conveyor_module_8_value_1 : INT;
	conveyor_module_8_value_2 : INT;
	conveyor_module_8_value_3 : INT;
	conveyor_module_8_value_4 : INT;
	conveyor_module_9_value_1 : INT;
	conveyor_module_9_value_2 : INT;
	conveyor_module_9_value_3 : INT;
	conveyor_module_9_value_4 : INT;
	conveyor_module_10_value_1 : INT;
	conveyor_module_10_value_2 : INT;
	conveyor_module_10_value_3 : INT;
	conveyor_module_10_value_4 : INT;
	conveyor_module_11_value_1 : INT;
	conveyor_module_11_value_2 : INT;
	conveyor_module_11_value_3 : INT;
	conveyor_module_11_value_4 : INT;
	conveyor_module_12_value_1 : INT;
	conveyor_module_12_value_2 : INT;
	conveyor_module_12_value_3 : INT;
	conveyor_module_12_value_4 : INT;
	conveyor_module_13_value_1 : INT;
	conveyor_module_13_value_2 : INT;
	conveyor_module_13_value_3 : INT;
	conveyor_module_13_value_4 : INT;
	conveyor_module_14_value_1 : INT;
	conveyor_module_14_value_2 : INT;
	conveyor_module_14_value_3 : INT;
	conveyor_module_14_value_4 : INT;
	conveyor_module_15_value_1 : INT;
	conveyor_module_15_value_2 : INT;
	conveyor_module_15_value_3 : INT;
	conveyor_module_15_value_4 : INT;
	conveyor_module_16_value_1 : INT;
	conveyor_module_16_value_2 : INT;
	conveyor_module_16_value_3 : INT;
	conveyor_module_16_value_4 : INT;
	conveyor_module_17_value_1 : INT;
	conveyor_module_17_value_2 : INT;
	conveyor_module_17_value_3 : INT;
	conveyor_module_17_value_4 : INT;
	conveyor_module_18_value_1 : INT;
	conveyor_module_18_value_2 : INT;
	conveyor_module_18_value_3 : INT;
	conveyor_module_18_value_4 : INT;
	conveyor_module_19_value_1 : INT;
	conveyor_module_19_value_2 : INT;
	conveyor_module_19_value_3 : INT;
	conveyor_module_19_value_4 : INT;
	conveyor_module_20_value_1 : INT;
	conveyor_module_20_value_2 : INT;
	conveyor_module_20_value_3 : INT;
	conveyor_module_20_value_4 : INT;
	conveyor_module_21_value_1 : INT;
	conveyor_module_21_value_2 : INT;
	conveyor_module_21_value_3 : INT;
	conveyor_module_21_value_4 : INT;
	conveyor_module_22_value_1 : INT;
	conveyor_module_22_value_2 : INT;
	conveyor_module_22_value_3 : INT;
	conveyor_module_22_value_4 : INT;
	conveyor_module_23_value_1 : INT;
	conveyor_module_23_value_2 : INT;
	conveyor_module_23_value_3 : INT;
	conveyor_module_23_value_4 : INT;
	conveyor_module_24_value_1 : INT;
	conveyor_module_24_value_2 : INT;
	conveyor_module_24_value_3 : INT;
	conveyor_module_24_value_4 : INT;
	conveyor_stop_word_1 : WORD;
	conveyor_stop_word_2 : WORD;
	conveyor_stop_word_3 : WORD;
	run_conveyor_1_fwd : BOOL;
	run_conveyor_1_rev : BOOL;
	conveyor_running_1 : BOOL;
	start_conveyor_1 : BOOL;
	stop_conveyor_1 : BOOL;
	estop_conveyor_1 : BOOL;
	want1 : BOOL;
	conveyor_stop_1 : BOOL;
	run_conveyor_2_fwd : BOOL;
	run_conveyor_2_rev : BOOL;
	conveyor_running_2 : BOOL;
	start_conveyor_2 : BOOL;
	stop_conveyor_2 : BOOL;
	estop_conveyor_2 : BOOL;
	want2 : BOOL;
	conveyor_stop_2 : BOOL;
	run_conveyor_3_fwd : BOOL;
	run_conveyor_3_rev : BOOL;
	conveyor_running_3 : BOOL;
	start_conveyor_3 : BOOL;
	stop_conveyor_3 : BOOL;
	estop_conveyor_3 : BOOL;
	want3 : BOOL;
	conveyor_stop_3 : BOOL;
	run_conveyor_4_fwd : BOOL;
	run_conveyor_4_rev : BOOL;
	conveyor_running_4 : BOOL;
	start_conveyor_4 : BOOL;
	stop_conveyor_4 : BOOL;
	estop_conveyor_4 : BOOL;
	want4 : BOOL;
	conveyor_stop_4 : BOOL;
	xfer_62_ok : BOOL;
	conv_61_ok : BOOL;
	Conver_61_ClearTimer : TON;
	Conveyor_61_ClearTime : INT := 10000;
	conveyor_61_complete : BOOL;
	conveyor_61_xfer_62_not_allowed : BOOL;
	xfer_72_ok : BOOL;
	conv_62_ok : BOOL;
	Conver_62_ClearTimer : TON;
	Conveyor_62_ClearTime : INT := 10000;
	conveyor_62_complete : BOOL;
	conveyor_62_xfer_72_not_allowed : BOOL;
	xfer_64_ok : BOOL;
	conv_63_ok : BOOL;
	Conver_63_ClearTimer : TON;
	Conveyor_63_ClearTime : INT := 10000;
	conveyor_63_complete : BOOL;
	conveyor_63_xfer_64_not_allowed : BOOL;
	xfer_73_ok : BOOL;
	conv_64_ok : BOOL;
	Conver_64_ClearTimer : TON;
	Conveyor_64_ClearTime : INT := 10000;
	conveyor_64_complete : BOOL;
	conveyor_64_xfer_73_not_allowed : BOOL;
	xfer_69_ok : BOOL;
	conv_68_ok : BOOL;
	Conver_68_ClearTimer : TON;
	Conveyor_68_ClearTime : INT := 10000;
	conveyor_68_complete : BOOL;
	conveyor_68_xfer_69_not_allowed : BOOL;
	xfer_70_ok : BOOL;
	conv_69_ok : BOOL;
	Conver_69_ClearTimer : TON;
	Conveyor_69_ClearTime : INT := 10000;
	conveyor_69_complete : BOOL;
	conveyor_69_xfer_70_not_allowed : BOOL;
	xfer_63_ok : BOOL;
	conv_70_ok : BOOL;
	Conver_70_ClearTimer : TON;
	Conveyor_70_ClearTime : INT := 10000;
	conveyor_70_complete : BOOL;
	conveyor_70_xfer_63_not_allowed : BOOL;
	xfer_66_ok : BOOL;
	conv_65_ok : BOOL;
	Conver_65_ClearTimer : TON;
	Conveyor_65_ClearTime : INT := 10000;
	conveyor_65_complete : BOOL;
	conveyor_65_xfer_66_not_allowed : BOOL;
	xfer_67_ok : BOOL;
	conv_66_ok : BOOL;
	Conver_66_ClearTimer : TON;
	Conveyor_66_ClearTime : INT := 10000;
	conveyor_66_complete : BOOL;
	conveyor_66_xfer_67_not_allowed : BOOL;
	xfer_61_ok : BOOL;
	conv_67_ok : BOOL;
	Conver_67_ClearTimer : TON;
	Conveyor_67_ClearTime : INT := 10000;
	conveyor_67_complete : BOOL;
	conveyor_67_xfer_61_not_allowed : BOOL;
	PANEL_ONLINE_1 : INT;
	weight1 : UINT;
	capture_weight_1 : UINT;
	min_weight_1 : UINT;
	near_weight_1 : UINT;
	buffer_weight_1 : UINT;
	notify_weight_1 : UINT;
	send_weight_1 : UINT;
	over_weight_1 : UINT;
	tare_value_1 : UINT;
	span_value_1 : UINT;
	myRaw1 : DINT;
	weight2 : UINT;
	capture_weight_2 : UINT;
	min_weight_2 : UINT;
	near_weight_2 : UINT;
	buffer_weight_2 : UINT;
	notify_weight_2 : UINT;
	send_weight_2 : UINT;
	over_weight_2 : UINT;
	tare_value_2 : UINT;
	span_value_2 : UINT;
	myRaw2 : DINT;
	weight3 : UINT;
	capture_weight_3 : UINT;
	min_weight_3 : UINT;
	near_weight_3 : UINT;
	buffer_weight_3 : UINT;
	notify_weight_3 : UINT;
	send_weight_3 : UINT;
	over_weight_3 : UINT;
	tare_value_3 : UINT;
	span_value_3 : UINT;
	myRaw3 : DINT;
	weight4 : UINT;
	capture_weight_4 : UINT;
	min_weight_4 : UINT;
	near_weight_4 : UINT;
	buffer_weight_4 : UINT;
	notify_weight_4 : UINT;
	send_weight_4 : UINT;
	over_weight_4 : UINT;
	tare_value_4 : UINT;
	span_value_4 : UINT;
	myRaw4 : DINT;
	weight5 : UINT;
	capture_weight_5 : UINT;
	min_weight_5 : UINT;
	near_weight_5 : UINT;
	buffer_weight_5 : UINT;
	notify_weight_5 : UINT;
	send_weight_5 : UINT;
	over_weight_5 : UINT;
	tare_value_5 : UINT;
	span_value_5 : UINT;
	myRaw5 : DINT;
	weight6 : UINT;
	capture_weight_6 : UINT;
	min_weight_6 : UINT;
	near_weight_6 : UINT;
	buffer_weight_6 : UINT;
	notify_weight_6 : UINT;
	send_weight_6 : UINT;
	over_weight_6 : UINT;
	tare_value_6 : UINT;
	span_value_6 : UINT;
	myRaw6 : DINT;
	weight7 : UINT;
	capture_weight_7 : UINT;
	min_weight_7 : UINT;
	near_weight_7 : UINT;
	buffer_weight_7 : UINT;
	notify_weight_7 : UINT;
	send_weight_7 : UINT;
	over_weight_7 : UINT;
	tare_value_7 : UINT;
	span_value_7 : UINT;
	myRaw7 : DINT;
	weight8 : UINT;
	capture_weight_8 : UINT;
	min_weight_8 : UINT;
	near_weight_8 : UINT;
	buffer_weight_8 : UINT;
	notify_weight_8 : UINT;
	send_weight_8 : UINT;
	over_weight_8 : UINT;
	tare_value_8 : UINT;
	span_value_8 : UINT;
	myRaw8 : DINT;
	weight9 : UINT;
	capture_weight_9 : UINT;
	min_weight_9 : UINT;
	near_weight_9 : UINT;
	buffer_weight_9 : UINT;
	notify_weight_9 : UINT;
	send_weight_9 : UINT;
	over_weight_9 : UINT;
	tare_value_9 : UINT;
	span_value_9 : UINT;
	myRaw9 : DINT;
	weight10 : UINT;
	capture_weight_10 : UINT;
	min_weight_10 : UINT;
	near_weight_10 : UINT;
	buffer_weight_10 : UINT;
	notify_weight_10 : UINT;
	send_weight_10 : UINT;
	over_weight_10 : UINT;
	tare_value_10 : UINT;
	span_value_10 : UINT;
	myRaw10 : DINT;
	weight11 : UINT;
	capture_weight_11 : UINT;
	min_weight_11 : UINT;
	near_weight_11 : UINT;
	buffer_weight_11 : UINT;
	notify_weight_11 : UINT;
	send_weight_11 : UINT;
	over_weight_11 : UINT;
	tare_value_11 : UINT;
	span_value_11 : UINT;
	myRaw11 : DINT;
	weight12 : UINT;
	capture_weight_12 : UINT;
	min_weight_12 : UINT;
	near_weight_12 : UINT;
	buffer_weight_12 : UINT;
	notify_weight_12 : UINT;
	send_weight_12 : UINT;
	over_weight_12 : UINT;
	tare_value_12 : UINT;
	span_value_12 : UINT;
	myRaw12 : DINT;
	weight13 : UINT;
	capture_weight_13 : UINT;
	min_weight_13 : UINT;
	near_weight_13 : UINT;
	buffer_weight_13 : UINT;
	notify_weight_13 : UINT;
	send_weight_13 : UINT;
	over_weight_13 : UINT;
	tare_value_13 : UINT;
	span_value_13 : UINT;
	myRaw13 : DINT;
	weight14 : UINT;
	capture_weight_14 : UINT;
	min_weight_14 : UINT;
	near_weight_14 : UINT;
	buffer_weight_14 : UINT;
	notify_weight_14 : UINT;
	send_weight_14 : UINT;
	over_weight_14 : UINT;
	tare_value_14 : UINT;
	span_value_14 : UINT;
	myRaw14 : DINT;
	weight15 : UINT;
	capture_weight_15 : UINT;
	min_weight_15 : UINT;
	near_weight_15 : UINT;
	buffer_weight_15 : UINT;
	notify_weight_15 : UINT;
	send_weight_15 : UINT;
	over_weight_15 : UINT;
	tare_value_15 : UINT;
	span_value_15 : UINT;
	myRaw15 : DINT;
	weight16 : UINT;
	capture_weight_16 : UINT;
	min_weight_16 : UINT;
	near_weight_16 : UINT;
	buffer_weight_16 : UINT;
	notify_weight_16 : UINT;
	send_weight_16 : UINT;
	over_weight_16 : UINT;
	tare_value_16 : UINT;
	span_value_16 : UINT;
	myRaw16 : DINT;
	weight17 : UINT;
	capture_weight_17 : UINT;
	min_weight_17 : UINT;
	near_weight_17 : UINT;
	buffer_weight_17 : UINT;
	notify_weight_17 : UINT;
	send_weight_17 : UINT;
	over_weight_17 : UINT;
	tare_value_17 : UINT;
	span_value_17 : UINT;
	myRaw17 : DINT;
	weight18 : UINT;
	capture_weight_18 : UINT;
	min_weight_18 : UINT;
	near_weight_18 : UINT;
	buffer_weight_18 : UINT;
	notify_weight_18 : UINT;
	send_weight_18 : UINT;
	over_weight_18 : UINT;
	tare_value_18 : UINT;
	span_value_18 : UINT;
	myRaw18 : DINT;
	weight19 : UINT;
	capture_weight_19 : UINT;
	min_weight_19 : UINT;
	near_weight_19 : UINT;
	buffer_weight_19 : UINT;
	notify_weight_19 : UINT;
	send_weight_19 : UINT;
	over_weight_19 : UINT;
	tare_value_19 : UINT;
	span_value_19 : UINT;
	myRaw19 : DINT;
	weight20 : UINT;
	capture_weight_20 : UINT;
	min_weight_20 : UINT;
	near_weight_20 : UINT;
	buffer_weight_20 : UINT;
	notify_weight_20 : UINT;
	send_weight_20 : UINT;
	over_weight_20 : UINT;
	tare_value_20 : UINT;
	span_value_20 : UINT;
	myRaw20 : DINT;
	weight21 : UINT;
	capture_weight_21 : UINT;
	min_weight_21 : UINT;
	near_weight_21 : UINT;
	buffer_weight_21 : UINT;
	notify_weight_21 : UINT;
	send_weight_21 : UINT;
	over_weight_21 : UINT;
	tare_value_21 : UINT;
	span_value_21 : UINT;
	myRaw21 : DINT;
	weight22 : UINT;
	capture_weight_22 : UINT;
	min_weight_22 : UINT;
	near_weight_22 : UINT;
	buffer_weight_22 : UINT;
	notify_weight_22 : UINT;
	send_weight_22 : UINT;
	over_weight_22 : UINT;
	tare_value_22 : UINT;
	span_value_22 : UINT;
	myRaw22 : DINT;
	weight23 : UINT;
	capture_weight_23 : UINT;
	min_weight_23 : UINT;
	near_weight_23 : UINT;
	buffer_weight_23 : UINT;
	notify_weight_23 : UINT;
	send_weight_23 : UINT;
	over_weight_23 : UINT;
	tare_value_23 : UINT;
	span_value_23 : UINT;
	myRaw23 : DINT;
	weight24 : UINT;
	capture_weight_24 : UINT;
	min_weight_24 : UINT;
	near_weight_24 : UINT;
	buffer_weight_24 : UINT;
	notify_weight_24 : UINT;
	send_weight_24 : UINT;
	over_weight_24 : UINT;
	tare_value_24 : UINT;
	span_value_24 : UINT;
	myRaw24 : DINT;
	weight25 : UINT;
	capture_weight_25 : UINT;
	min_weight_25 : UINT;
	near_weight_25 : UINT;
	buffer_weight_25 : UINT;
	notify_weight_25 : UINT;
	send_weight_25 : UINT;
	over_weight_25 : UINT;
	tare_value_25 : UINT;
	span_value_25 : UINT;
	myRaw25 : DINT;
	weight26 : UINT;
	capture_weight_26 : UINT;
	min_weight_26 : UINT;
	near_weight_26 : UINT;
	buffer_weight_26 : UINT;
	notify_weight_26 : UINT;
	send_weight_26 : UINT;
	over_weight_26 : UINT;
	tare_value_26 : UINT;
	span_value_26 : UINT;
	myRaw26 : DINT;
	weight27 : UINT;
	capture_weight_27 : UINT;
	min_weight_27 : UINT;
	near_weight_27 : UINT;
	buffer_weight_27 : UINT;
	notify_weight_27 : UINT;
	send_weight_27 : UINT;
	over_weight_27 : UINT;
	tare_value_27 : UINT;
	span_value_27 : UINT;
	myRaw27 : DINT;
	weight28 : UINT;
	capture_weight_28 : UINT;
	min_weight_28 : UINT;
	near_weight_28 : UINT;
	buffer_weight_28 : UINT;
	notify_weight_28 : UINT;
	send_weight_28 : UINT;
	over_weight_28 : UINT;
	tare_value_28 : UINT;
	span_value_28 : UINT;
	myRaw28 : DINT;
	weight29 : UINT;
	capture_weight_29 : UINT;
	min_weight_29 : UINT;
	near_weight_29 : UINT;
	buffer_weight_29 : UINT;
	notify_weight_29 : UINT;
	send_weight_29 : UINT;
	over_weight_29 : UINT;
	tare_value_29 : UINT;
	span_value_29 : UINT;
	myRaw29 : DINT;
	weight30 : UINT;
	capture_weight_30 : UINT;
	min_weight_30 : UINT;
	near_weight_30 : UINT;
	buffer_weight_30 : UINT;
	notify_weight_30 : UINT;
	send_weight_30 : UINT;
	over_weight_30 : UINT;
	tare_value_30 : UINT;
	span_value_30 : UINT;
	myRaw30 : DINT;
	weight31 : UINT;
	capture_weight_31 : UINT;
	min_weight_31 : UINT;
	near_weight_31 : UINT;
	buffer_weight_31 : UINT;
	notify_weight_31 : UINT;
	send_weight_31 : UINT;
	over_weight_31 : UINT;
	tare_value_31 : UINT;
	span_value_31 : UINT;
	myRaw31 : DINT;
	weight32 : UINT;
	capture_weight_32 : UINT;
	min_weight_32 : UINT;
	near_weight_32 : UINT;
	buffer_weight_32 : UINT;
	notify_weight_32 : UINT;
	send_weight_32 : UINT;
	over_weight_32 : UINT;
	tare_value_32 : UINT;
	span_value_32 : UINT;
	myRaw32 : DINT;
	weight33 : UINT;
	capture_weight_33 : UINT;
	min_weight_33 : UINT;
	near_weight_33 : UINT;
	buffer_weight_33 : UINT;
	notify_weight_33 : UINT;
	send_weight_33 : UINT;
	over_weight_33 : UINT;
	tare_value_33 : UINT;
	span_value_33 : UINT;
	myRaw33 : DINT;
	weight34 : UINT;
	capture_weight_34 : UINT;
	min_weight_34 : UINT;
	near_weight_34 : UINT;
	buffer_weight_34 : UINT;
	notify_weight_34 : UINT;
	send_weight_34 : UINT;
	over_weight_34 : UINT;
	tare_value_34 : UINT;
	span_value_34 : UINT;
	myRaw34 : DINT;
	weight35 : UINT;
	capture_weight_35 : UINT;
	min_weight_35 : UINT;
	near_weight_35 : UINT;
	buffer_weight_35 : UINT;
	notify_weight_35 : UINT;
	send_weight_35 : UINT;
	over_weight_35 : UINT;
	tare_value_35 : UINT;
	span_value_35 : UINT;
	myRaw35 : DINT;
	weight36 : UINT;
	capture_weight_36 : UINT;
	min_weight_36 : UINT;
	near_weight_36 : UINT;
	buffer_weight_36 : UINT;
	notify_weight_36 : UINT;
	send_weight_36 : UINT;
	over_weight_36 : UINT;
	tare_value_36 : UINT;
	span_value_36 : UINT;
	myRaw36 : DINT;
	weight37 : UINT;
	capture_weight_37 : UINT;
	min_weight_37 : UINT;
	near_weight_37 : UINT;
	buffer_weight_37 : UINT;
	notify_weight_37 : UINT;
	send_weight_37 : UINT;
	over_weight_37 : UINT;
	tare_value_37 : UINT;
	span_value_37 : UINT;
	myRaw37 : DINT;
	weight38 : UINT;
	capture_weight_38 : UINT;
	min_weight_38 : UINT;
	near_weight_38 : UINT;
	buffer_weight_38 : UINT;
	notify_weight_38 : UINT;
	send_weight_38 : UINT;
	over_weight_38 : UINT;
	tare_value_38 : UINT;
	span_value_38 : UINT;
	myRaw38 : DINT;
	weight39 : UINT;
	capture_weight_39 : UINT;
	min_weight_39 : UINT;
	near_weight_39 : UINT;
	buffer_weight_39 : UINT;
	notify_weight_39 : UINT;
	send_weight_39 : UINT;
	over_weight_39 : UINT;
	tare_value_39 : UINT;
	span_value_39 : UINT;
	myRaw39 : DINT;
	weight40 : UINT;
	capture_weight_40 : UINT;
	min_weight_40 : UINT;
	near_weight_40 : UINT;
	buffer_weight_40 : UINT;
	notify_weight_40 : UINT;
	send_weight_40 : UINT;
	over_weight_40 : UINT;
	tare_value_40 : UINT;
	span_value_40 : UINT;
	myRaw40 : DINT;
	weight41 : UINT;
	capture_weight_41 : UINT;
	min_weight_41 : UINT;
	near_weight_41 : UINT;
	buffer_weight_41 : UINT;
	notify_weight_41 : UINT;
	send_weight_41 : UINT;
	over_weight_41 : UINT;
	tare_value_41 : UINT;
	span_value_41 : UINT;
	myRaw41 : DINT;
	weight42 : UINT;
	capture_weight_42 : UINT;
	min_weight_42 : UINT;
	near_weight_42 : UINT;
	buffer_weight_42 : UINT;
	notify_weight_42 : UINT;
	send_weight_42 : UINT;
	over_weight_42 : UINT;
	tare_value_42 : UINT;
	span_value_42 : UINT;
	myRaw42 : DINT;
	weight43 : UINT;
	capture_weight_43 : UINT;
	min_weight_43 : UINT;
	near_weight_43 : UINT;
	buffer_weight_43 : UINT;
	notify_weight_43 : UINT;
	send_weight_43 : UINT;
	over_weight_43 : UINT;
	tare_value_43 : UINT;
	span_value_43 : UINT;
	myRaw43 : DINT;
	weight44 : UINT;
	capture_weight_44 : UINT;
	min_weight_44 : UINT;
	near_weight_44 : UINT;
	buffer_weight_44 : UINT;
	notify_weight_44 : UINT;
	send_weight_44 : UINT;
	over_weight_44 : UINT;
	tare_value_44 : UINT;
	span_value_44 : UINT;
	myRaw44 : DINT;
	weight45 : UINT;
	capture_weight_45 : UINT;
	min_weight_45 : UINT;
	near_weight_45 : UINT;
	buffer_weight_45 : UINT;
	notify_weight_45 : UINT;
	send_weight_45 : UINT;
	over_weight_45 : UINT;
	tare_value_45 : UINT;
	span_value_45 : UINT;
	myRaw45 : DINT;
	weight46 : UINT;
	capture_weight_46 : UINT;
	min_weight_46 : UINT;
	near_weight_46 : UINT;
	buffer_weight_46 : UINT;
	notify_weight_46 : UINT;
	send_weight_46 : UINT;
	over_weight_46 : UINT;
	tare_value_46 : UINT;
	span_value_46 : UINT;
	myRaw46 : DINT;
	weight47 : UINT;
	capture_weight_47 : UINT;
	min_weight_47 : UINT;
	near_weight_47 : UINT;
	buffer_weight_47 : UINT;
	notify_weight_47 : UINT;
	send_weight_47 : UINT;
	over_weight_47 : UINT;
	tare_value_47 : UINT;
	span_value_47 : UINT;
	myRaw47 : DINT;
	weight48 : UINT;
	capture_weight_48 : UINT;
	min_weight_48 : UINT;
	near_weight_48 : UINT;
	buffer_weight_48 : UINT;
	notify_weight_48 : UINT;
	send_weight_48 : UINT;
	over_weight_48 : UINT;
	tare_value_48 : UINT;
	span_value_48 : UINT;
	myRaw48 : DINT;
	weight49 : UINT;
	capture_weight_49 : UINT;
	min_weight_49 : UINT;
	near_weight_49 : UINT;
	buffer_weight_49 : UINT;
	notify_weight_49 : UINT;
	send_weight_49 : UINT;
	over_weight_49 : UINT;
	tare_value_49 : UINT;
	span_value_49 : UINT;
	myRaw49 : DINT;
	weight50 : UINT;
	capture_weight_50 : UINT;
	min_weight_50 : UINT;
	near_weight_50 : UINT;
	buffer_weight_50 : UINT;
	notify_weight_50 : UINT;
	send_weight_50 : UINT;
	over_weight_50 : UINT;
	tare_value_50 : UINT;
	span_value_50 : UINT;
	myRaw50 : DINT;
	weight51 : UINT;
	capture_weight_51 : UINT;
	min_weight_51 : UINT;
	near_weight_51 : UINT;
	buffer_weight_51 : UINT;
	notify_weight_51 : UINT;
	send_weight_51 : UINT;
	over_weight_51 : UINT;
	tare_value_51 : UINT;
	span_value_51 : UINT;
	myRaw51 : DINT;
	weight52 : UINT;
	capture_weight_52 : UINT;
	min_weight_52 : UINT;
	near_weight_52 : UINT;
	buffer_weight_52 : UINT;
	notify_weight_52 : UINT;
	send_weight_52 : UINT;
	over_weight_52 : UINT;
	tare_value_52 : UINT;
	span_value_52 : UINT;
	myRaw52 : DINT;
	weight53 : UINT;
	capture_weight_53 : UINT;
	min_weight_53 : UINT;
	near_weight_53 : UINT;
	buffer_weight_53 : UINT;
	notify_weight_53 : UINT;
	send_weight_53 : UINT;
	over_weight_53 : UINT;
	tare_value_53 : UINT;
	span_value_53 : UINT;
	myRaw53 : DINT;
	weight54 : UINT;
	capture_weight_54 : UINT;
	min_weight_54 : UINT;
	near_weight_54 : UINT;
	buffer_weight_54 : UINT;
	notify_weight_54 : UINT;
	send_weight_54 : UINT;
	over_weight_54 : UINT;
	tare_value_54 : UINT;
	span_value_54 : UINT;
	myRaw54 : DINT;
	weight55 : UINT;
	capture_weight_55 : UINT;
	min_weight_55 : UINT;
	near_weight_55 : UINT;
	buffer_weight_55 : UINT;
	notify_weight_55 : UINT;
	send_weight_55 : UINT;
	over_weight_55 : UINT;
	tare_value_55 : UINT;
	span_value_55 : UINT;
	myRaw55 : DINT;
	weight56 : UINT;
	capture_weight_56 : UINT;
	min_weight_56 : UINT;
	near_weight_56 : UINT;
	buffer_weight_56 : UINT;
	notify_weight_56 : UINT;
	send_weight_56 : UINT;
	over_weight_56 : UINT;
	tare_value_56 : UINT;
	span_value_56 : UINT;
	myRaw56 : DINT;
	weight57 : UINT;
	capture_weight_57 : UINT;
	min_weight_57 : UINT;
	near_weight_57 : UINT;
	buffer_weight_57 : UINT;
	notify_weight_57 : UINT;
	send_weight_57 : UINT;
	over_weight_57 : UINT;
	tare_value_57 : UINT;
	span_value_57 : UINT;
	myRaw57 : DINT;
	weight58 : UINT;
	capture_weight_58 : UINT;
	min_weight_58 : UINT;
	near_weight_58 : UINT;
	buffer_weight_58 : UINT;
	notify_weight_58 : UINT;
	send_weight_58 : UINT;
	over_weight_58 : UINT;
	tare_value_58 : UINT;
	span_value_58 : UINT;
	myRaw58 : DINT;
	weight59 : UINT;
	capture_weight_59 : UINT;
	min_weight_59 : UINT;
	near_weight_59 : UINT;
	buffer_weight_59 : UINT;
	notify_weight_59 : UINT;
	send_weight_59 : UINT;
	over_weight_59 : UINT;
	tare_value_59 : UINT;
	span_value_59 : UINT;
	myRaw59 : DINT;
	weight60 : UINT;
	capture_weight_60 : UINT;
	min_weight_60 : UINT;
	near_weight_60 : UINT;
	buffer_weight_60 : UINT;
	notify_weight_60 : UINT;
	send_weight_60 : UINT;
	over_weight_60 : UINT;
	tare_value_60 : UINT;
	span_value_60 : UINT;
	myRaw60 : DINT;
	loadcell_array : ARRAY[0..60] OF LoadCell;
	loadcell_udp_array : ARRAY[0..60] OF LoadcellUdpType;
	io_comm : ARRAY[0..0] OF WORD;
	insert_reset_1 : WORD;
	waiting_1 : WORD;
	insert_1 : WORD;
	bring_ok_1 : WORD;
	alarm_1 : WORD;
	insert_reset_2 : WORD;
	waiting_2 : WORD;
	insert_2 : WORD;
	bring_ok_2 : WORD;
	alarm_2 : WORD;
	insert_reset_3 : WORD;
	waiting_3 : WORD;
	insert_3 : WORD;
	bring_ok_3 : WORD;
	alarm_3 : WORD;
	insert_reset_4 : WORD;
	waiting_4 : WORD;
	insert_4 : WORD;
	bring_ok_4 : WORD;
	alarm_4 : WORD;
	insert_reset_5 : WORD;
	waiting_5 : WORD;
	insert_5 : WORD;
	bring_ok_5 : WORD;
	alarm_5 : WORD;
	rail_destination_1 : INT;
	rail_destination_2 : INT;
	rail_destination_3 : INT;
	rail_destination_4 : INT;
	rail_destination_5 : INT;
	rail_destination_6 : INT;
	rail_destination_7 : INT;
	rail_destination_8 : INT;
	rail_destination_9 : INT;
	rail_destination_10 : INT;
	rail_destination_11 : INT;
	rail_destination_12 : INT;
	rail_destination_13 : INT;
	rail_destination_14 : INT;
	rail_destination_15 : INT;
	rail_destination_16 : INT;
	rail_destination_17 : INT;
	rail_destination_18 : INT;
	rail_destination_19 : INT;
	rail_destination_20 : INT;
	rail_destination_21 : INT;
	rail_destination_22 : INT;
	rail_destination_23 : INT;
	rail_destination_24 : INT;
	rail_destination_25 : INT;
	rail_destination_26 : INT;
	rail_destination_27 : INT;
	rail_destination_28 : INT;
	rail_destination_29 : INT;
	rail_destination_30 : INT;
	rail_destination_31 : INT;
	rail_destination_32 : INT;
	rail_destination_33 : INT;
	rail_destination_34 : INT;
	rail_destination_35 : INT;
	rail_destination_36 : INT;
	rail_destination_37 : INT;
	rail_destination_38 : INT;
	rail_destination_39 : INT;
	rail_destination_40 : INT;
	rail_destination_41 : INT;
	rail_destination_42 : INT;
	rail_destination_43 : INT;
	rail_destination_44 : INT;
	rail_destination_45 : INT;
	rail_destination_46 : INT;
	rail_destination_47 : INT;
	rail_destination_48 : INT;
	rail_destination_49 : INT;
	rail_destination_50 : INT;
	rail_destination_51 : INT;
	rail_destination_52 : INT;
	rail_destination_53 : INT;
	rail_destination_54 : INT;
	rail_destination_55 : INT;
	rail_destination_56 : INT;
	rail_destination_57 : INT;
	rail_destination_58 : INT;
	rail_destination_59 : INT;
	rail_destination_60 : INT;
	rail_destination_61 : INT;
	rail_destination_62 : INT;
	rail_destination_63 : INT;
	rail_destination_64 : INT;
	rail_destination_65 : INT;
	rail_destination_66 : INT;
	rail_destination_67 : INT;
	rail_destination_68 : INT;
	rail_destination_69 : INT;
	rail_destination_70 : INT;
	rail_destination_71 : INT;
	rail_destination_72 : INT;
	rail_destination_73 : INT;
	rail_destination_74 : INT;
	rail_destination_75 : INT;
	rail_destination_76 : INT;
	rail_destination_77 : INT;
	rail_destination_78 : INT;
	rail_destination_79 : INT;
	rail_destination_80 : INT;
	rail_destination_81 : INT;
	rail_destination_82 : INT;
	rail_destination_83 : INT;
	rail_destination_84 : INT;
	rail_destination_85 : INT;
	rail_destination_86 : INT;
	rail_destination_87 : INT;
	rail_destination_88 : INT;
	rail_destination_89 : INT;
	rail_destination_90 : INT;
	rail_destination_91 : INT;
	rail_destination_92 : INT;
	rail_destination_93 : INT;
	rail_destination_94 : INT;
	rail_destination_95 : INT;
	rail_destination_96 : INT;
	rail_destination_97 : INT;
	rail_destination_98 : INT;
	rail_destination_99 : INT;
	rail_destination_100 : INT;
	rail_destination_101 : INT;
	DEST_SIZE : INT;
	DEST_NUM : INT;
	DEST_RAIL : INT;
	DEST_INDEX : INT;
	bank_1_clear : BOOL;
	bank_1_clear_timer : TON;
	bank_4_clear : BOOL;
	bank_4_clear_timer : TON;
	bank_5_clear : BOOL;
	bank_5_clear_timer : TON;
	bank_6_clear : BOOL;
	bank_6_clear_timer : TON;
	bank_2_clear : BOOL;
	bank_2_clear_timer : TON;
	bank_3_clear : BOOL;
	bank_3_clear_timer : TON;
END_VAR
```

### Custom_Variables.var
```iecst
VAR
	CC_EStop_Safety : BOOL;
	customTest : BOOL;
	EStop : ARRAY[1..4] OF BOOL;
	Fuse_Lamp_1 : BOOL;
	Fuse_Lamp_2 : BOOL;
	Fuse_Lamp_3 : BOOL;
	Fuse_Reset_1 : BOOL;
	Fuse_Reset_2 : BOOL;
	Fuse_Reset_3 : BOOL;
END_VAR
VAR RETAIN
	gEmptyLine : {REDUND_UNREPLICABLE} BOOL;
END_VAR
VAR
	MasterReset_1 : BOOL;
	MasterReset_2 : BOOL;
	MasterReset_3 : BOOL;
	MasterReset_MC01 : BOOL;
	Fuse_Reset_MC01 : BOOL;
	MasterReset_MC02 : BOOL;
	Fuse_Reset_MC02 : BOOL;
	sb1_endPX : BOOL;
	sb1_lamp : BOOL;
	sb1_start : BOOL;
	sb1_stop : BOOL;
	sb2_endPX : BOOL;
	sb3_endPX : BOOL;
	sb2_start : BOOL;
	sb2_stop : BOOL;
	sb2_lamp : BOOL;
	pressure_sensor1 : BOOL;
	pressure_sensor2 : BOOL;
	tripCurrent : USINT;
	SSL2_LowerGuard : BOOL;
	SSL2_RaiseGuard : BOOL;
	ssr1_prs : BOOL;
	ssr1_close : BOOL;
END_VAR
```

### Program Logical/DBOUNCE (IEC, version 1.00.1) - DBOUNCE

#### DBOUNCE.st
```iecst
(********************************************************************
 * Program: dbounce
 * File: dbounce.st
 ********************************************************************)
PROGRAM _CYCLIC
	(* Pulse Generators *)
	one_sec_pulse(IN:= not_one_sec_pulse.Q, PT:= t#1s);
	not_one_sec_pulse(IN:=NOT(one_sec_pulse.Q), PT:= t#1s);
	thirty_msec_pulse(IN:= not_thirty_msec_pulse.Q, PT:= t#30ms);
	not_thirty_msec_pulse(IN:=NOT(thirty_msec_pulse.Q), PT:= t#30ms);

END_PROGRAM
```

### Program Logical/ALARMS (IEC, version 1.00.1) - ALARMS
